LIN {X 0,Y 155.826,Z 845.987,A -85,B 0,C 180,E1 -23873.947,E2 -23873.947} C_VEL
LIN {X 0,Y 159.588,Z 842.317,A -85,B 0,C 180,E1 -23877.541,E2 -23877.541} C_VEL
LIN {X 0,Y 163.776,Z 837.68,A -85,B 0,C 180,E1 -23880.992,E2 -23880.992} C_VEL
LIN {X 0,Y 169.657,Z 830.821,A -85,B 0,C 180,E1 -23884.72,E2 -23884.72} C_VEL
LIN {X 0,Y 175.318,Z 823.487,A -85,B 0,C 180,E1 -23887.684,E2 -23887.684} C_VEL
LIN {X 0,Y 181.515,Z 814.528,A -85,B 0,C 180,E1 -23890.429,E2 -23890.429} C_VEL
LIN {X 0,Y 186.46,Z 805.713,A -85,B 0,C 180,E1 -23892.721,E2 -23892.721} C_VEL
LIN {X 0,Y 191.129,Z 795.722,A -85,B 0,C 180,E1 -23894.904,E2 -23894.904} C_VEL
LIN {X 0,Y 194.213,Z 785.837,A -85,B 0,C 180,E1 -23897.193,E2 -23897.193} C_VEL
LIN {X 0,Y 196.046,Z 776.648,A -85,B 0,C 180,E1 -23899.421,E2 -23899.421} C_VEL
LIN {X 0,Y 196.921,Z 769.856,A -85,B 0,C 180,E1 -23901.188,E2 -23901.188} C_VEL
LIN {X 0,Y 196.991,Z 768.155,A -85,B 0,C 180,E1 -23901.708,E2 -23901.708} C_VEL
LIN {X 0,Y 195.839,Z 762.077,A -85,B 0,C 180,E1 -23904.957,E2 -23904.957} C_VEL
LIN {X 0,Y 195.533,Z 760.977,A -85,B 0,C 180,E1 -23905.757,E2 -23905.757} C_VEL
LIN {X 0,Y 194.784,Z 759.757,A -85,B 0,C 180,E1 -23907.233,E2 -23907.233} C_VEL
LIN {X 0,Y 193.221,Z 757.907,A -85,B 0,C 180,E1 -23911.128,E2 -23911.128} C_VEL
LIN {X 0,Y 192.563,Z 757.534,A -85,B 0,C 180,E1 -23914.025,E2 -23914.025} C_VEL
LIN {X 0,Y 192.277,Z 757.927,A -85,B 0,C 180,E1 -23916.292,E2 -23916.292} C_VEL
LIN {X 0,Y 192.26,Z 758.818,A -85,B 0,C 180,E1 -23918.558,E2 -23918.558} C_VEL
LIN {X 0,Y 192.645,Z 760.564,A -85,B 0,C 180,E1 -23921.531,E2 -23921.531} C_VEL
LIN {X 0,Y 193.16,Z 762.881,A -85,B 0,C 180,E1 -23924.02,E2 -23924.02} C_VEL
LIN {X 0,Y 193.845,Z 765.735,A -85,B 0,C 180,E1 -23926.409,E2 -23926.409} C_VEL
LIN {X 0,Y 194.652,Z 771.052,A -85,B 0,C 180,E1 -23929.599,E2 -23929.599} C_VEL
LIN {X 0,Y 194.221,Z 775.457,A -85,B 0,C 180,E1 -23931.153,E2 -23931.153} C_VEL
LIN {X 0,Y 192.654,Z 785.131,A -85,B 0,C 180,E1 -23934.242,E2 -23934.242} C_VEL
LIN {X 0,Y 190.272,Z 794.462,A -85,B 0,C 180,E1 -23937.142,E2 -23937.142} C_VEL
LIN {X 0,Y 188.258,Z 800.26,A -85,B 0,C 180,E1 -23938.93,E2 -23938.93} C_VEL
LIN {X 0,Y 181.902,Z 810.719,A -85,B 0,C 180,E1 -23941.589,E2 -23941.589} C_VEL
LIN {X 0,Y 175.399,Z 819.674,A -85,B 0,C 180,E1 -23944.596,E2 -23944.596} C_VEL
LIN {X 0,Y 170.121,Z 826.215,A -85,B 0,C 180,E1 -23947.498,E2 -23947.498} C_VEL
LIN {X 0,Y 164.672,Z 832.219,A -85,B 0,C 180,E1 -23951.014,E2 -23951.014} C_VEL
LIN {X 0,Y 159.317,Z 837.423,A -85,B 0,C 180,E1 -23955.348,E2 -23955.348} C_VEL
LIN {X 0,Y 155.916,Z 840.355,A -85,B 0,C 180,E1 -23958.817,E2 -23958.817} C_VEL
LIN {X 0,Y 152.704,Z 842.697,A -85,B 0,C 180,E1 -23963.01,E2 -23963.01} C_VEL
LIN {X 0,Y 149.965,Z 844.066,A -85,B 0,C 180,E1 -23967.946,E2 -23967.946} C_VEL
LIN {X 0,Y 148.566,Z 844.232,A -85,B 0,C 180,E1 -23971.628,E2 -23971.628} C_VEL
LIN {X 0,Y 147.557,Z 843.519,A -85,B 0,C 180,E1 -23975.937,E2 -23975.937} C_VEL
LIN {X 0,Y 147.083,Z 841.894,A -85,B 0,C 180,E1 -23980.139,E2 -23980.139} C_VEL
LIN {X 0,Y 147.203,Z 839.369,A -85,B 0,C 180,E1 -23984.265,E2 -23984.265} C_VEL
LIN {X 0,Y 147.768,Z 835.966,A -85,B 0,C 180,E1 -23988.254,E2 -23988.254} C_VEL
LIN {X 0,Y 148.67,Z 831.692,A -85,B 0,C 180,E1 -23992.083,E2 -23992.083} C_VEL
LIN {X 0,Y 150.258,Z 825.225,A -85,B 0,C 180,E1 -23996.557,E2 -23996.557} C_VEL
LIN {X 0,Y 152.117,Z 818.304,A -85,B 0,C 180,E1 -24000.31,E2 -24000.31} C_VEL
LIN {X 0,Y 154.493,Z 809.866,A -85,B 0,C 180,E1 -24003.95,E2 -24003.95} C_VEL
LIN {X 0,Y 157.066,Z 800.56,A -85,B 0,C 180,E1 -24007.131,E2 -24007.131} C_VEL
LIN {X 0,Y 159.971,Z 789.532,A -85,B 0,C 180,E1 -24010.095,E2 -24010.095} C_VEL
LIN {X 0,Y 162.101,Z 780.609,A -85,B 0,C 180,E1 -24012.008,E2 -24012.008} C_VEL
LIN {X 0,Y 161.942,Z 769.581,A -85,B 0,C 180,E1 -24014.263,E2 -24014.263} C_VEL
LIN {X 0,Y 161.075,Z 757.75,A -85,B 0,C 180,E1 -24016.295,E2 -24016.295} C_VEL
LIN {X 0,Y 159.614,Z 744.505,A -85,B 0,C 180,E1 -24018.114,E2 -24018.114} C_VEL
LIN {X 0,Y 157.757,Z 732.883,A -85,B 0,C 180,E1 -24019.46,E2 -24019.46} C_VEL
LIN {X 0,Y 159.668,Z 724.11,A -85,B 0,C 180,E1 -24024.318,E2 -24024.318} C_VEL
LIN {X 0,Y 159.312,Z 719.069,A -85,B 0,C 180,E1 -24027.473,E2 -24027.473} C_VEL
LIN {X 0,Y 158.489,Z 711.374,A -85,B 0,C 180,E1 -24032.543,E2 -24032.543} C_VEL
LIN {X 0,Y 157.745,Z 708.301,A -85,B 0,C 180,E1 -24034.713,E2 -24034.713} C_VEL
LIN {X 0,Y 161.91,Z 713.53,A -85,B 0,C 180,E1 -24036.857,E2 -24036.857} C_VEL
LIN {X 0,Y 163.628,Z 720.985,A -85,B 0,C 180,E1 -24039.27,E2 -24039.27} C_VEL
LIN {X 0,Y 162.948,Z 724.437,A -85,B 0,C 180,E1 -24040.249,E2 -24040.249} C_VEL
LIN {X 0,Y 160.426,Z 733.712,A -85,B 0,C 180,E1 -24043.16,E2 -24043.16} C_VEL
LIN {X 0,Y 157.619,Z 743.025,A -85,B 0,C 180,E1 -24046.849,E2 -24046.849} C_VEL
LIN {X 0,Y 155.336,Z 750.632,A -85,B 0,C 180,E1 -24050.67,E2 -24050.67} C_VEL
LIN {X 0,Y 153.367,Z 757.474,A -85,B 0,C 180,E1 -24055.081,E2 -24055.081} C_VEL
LIN {X 0,Y 152.207,Z 761.853,A -85,B 0,C 180,E1 -24058.681,E2 -24058.681} C_VEL
LIN {X 0,Y 151.345,Z 766.086,A -85,B 0,C 180,E1 -24063.294,E2 -24063.294} C_VEL
LIN {X 0,Y 151.242,Z 768.983,A -85,B 0,C 180,E1 -24067.818,E2 -24067.818} C_VEL
LIN {X 0,Y 151.842,Z 770.706,A -85,B 0,C 180,E1 -24072.221,E2 -24072.221} C_VEL
LIN {X 0,Y 153.463,Z 771.373,A -85,B 0,C 180,E1 -24077.118,E2 -24077.118} C_VEL
LIN {X 0,Y 155.151,Z 770.994,A -85,B 0,C 180,E1 -24080.642,E2 -24080.642} C_VEL
LIN {X 0,Y 157.614,Z 769.708,A -85,B 0,C 180,E1 -24084.573,E2 -24084.573} C_VEL
LIN {X 0,Y 160.613,Z 767.497,A -85,B 0,C 180,E1 -24088.326,E2 -24088.326} C_VEL
LIN {X 0,Y 164.018,Z 764.381,A -85,B 0,C 180,E1 -24091.879,E2 -24091.879} C_VEL
LIN {X 0,Y 169.07,Z 758.981,A -85,B 0,C 180,E1 -24096.138,E2 -24096.138} C_VEL
LIN {X 0,Y 174.209,Z 752.578,A -85,B 0,C 180,E1 -24099.714,E2 -24099.714} C_VEL
LIN {X 0,Y 179.683,Z 744.584,A -85,B 0,C 180,E1 -24103.073,E2 -24103.073} C_VEL
LIN {X 0,Y 180.22,Z 740.718,A -85,B 0,C 180,E1 -24105.317,E2 -24105.317} C_VEL
LIN {X 0,Y 180.167,Z 735.06,A -85,B 0,C 180,E1 -24108.753,E2 -24108.753} C_VEL
LIN {X 0,Y 179.591,Z 729.771,A -85,B 0,C 180,E1 -24112.128,E2 -24112.128} C_VEL
LIN {X 0,Y 178.743,Z 724.926,A -85,B 0,C 180,E1 -24115.49,E2 -24115.49} C_VEL
LIN {X 0,Y 177.285,Z 719.37,A -85,B 0,C 180,E1 -24120,E2 -24120} C_VEL
LIN {X 0,Y 176.628,Z 716.866,A -85,B 0,C 180,E1 -24122.281,E2 -24122.281} C_VEL
LIN {X 0,Y 175.812,Z 715.036,A -85,B 0,C 180,E1 -24124.586,E2 -24124.586} C_VEL
LIN {X 0,Y 174.96,Z 713.779,A -85,B 0,C 180,E1 -24126.922,E2 -24126.922} C_VEL
LIN {X 0,Y 174.184,Z 713.013,A -85,B 0,C 180,E1 -24129.288,E2 -24129.288} C_VEL
LIN {X 0,Y 172.617,Z 713.732,A -85,B 0,C 180,E1 -24136.559,E2 -24136.559} C_VEL
LIN {X 0,Y 172.623,Z 715.509,A -85,B 0,C 180,E1 -24140.542,E2 -24140.542} C_VEL
LIN {X 0,Y 173.211,Z 719.303,A -85,B 0,C 180,E1 -24145.217,E2 -24145.217} C_VEL
LIN {X 0,Y 174.877,Z 724.229,A -85,B 0,C 180,E1 -24150.072,E2 -24150.072} C_VEL
LIN {X 0,Y 176.562,Z 731.034,A -85,B 0,C 180,E1 -24154.475,E2 -24154.475} C_VEL
LIN {X 0,Y 177.831,Z 737.369,A -85,B 0,C 180,E1 -24157.775,E2 -24157.775} C_VEL
LIN {X 0,Y 178.755,Z 742.992,A -85,B 0,C 180,E1 -24160.37,E2 -24160.37} C_VEL
LIN {X 0,Y 178.012,Z 748.71,A -85,B 0,C 180,E1 -24162.158,E2 -24162.158} C_VEL
LIN {X 0,Y 175.591,Z 759.813,A -85,B 0,C 180,E1 -24165.539,E2 -24165.539} C_VEL
LIN {X 0,Y 172.631,Z 769.223,A -85,B 0,C 180,E1 -24168.586,E2 -24168.586} C_VEL
LIN {X 0,Y 168.859,Z 778.701,A -85,B 0,C 180,E1 -24172.027,E2 -24172.027} C_VEL
LIN {X 0,Y 164.593,Z 786.996,A -85,B 0,C 180,E1 -24175.543,E2 -24175.543} C_VEL
LIN {X 0,Y 160.441,Z 794.744,A -85,B 0,C 180,E1 -24179.75,E2 -24179.75} C_VEL
LIN {X 0,Y 159.775,Z 795.982,A -85,B 0,C 180,E1 -24180.429,E2 -24180.429} C_VEL
LIN {X 0,Y 157.071,Z 806.36,A -85,B 0,C 180,E1 -24183.06,E2 -24183.06} C_VEL
LIN {X 0,Y 154.684,Z 815.135,A -85,B 0,C 180,E1 -24185.862,E2 -24185.862} C_VEL
LIN {X 0,Y 152.114,Z 824.713,A -85,B 0,C 180,E1 -24189.724,E2 -24189.724} C_VEL
LIN {X 0,Y 150.069,Z 832.34,A -85,B 0,C 180,E1 -24193.679,E2 -24193.679} C_VEL
LIN {X 0,Y 148.844,Z 838.458,A -85,B 0,C 180,E1 -24197.731,E2 -24197.731} C_VEL
LIN {X 0,Y 148.118,Z 843.259,A -85,B 0,C 180,E1 -24201.815,E2 -24201.815} C_VEL
LIN {X 0,Y 147.923,Z 845.823,A -85,B 0,C 180,E1 -24204.546,E2 -24204.546} C_VEL
LIN {X 0,Y 147.845,Z 847.879,A -85,B 0,C 180,E1 -24207.274,E2 -24207.274} C_VEL
LIN {X 0,Y 147.968,Z 849.477,A -85,B 0,C 180,E1 -24209.999,E2 -24209.999} C_VEL
LIN {X 0,Y 147.782,Z 851.409,A -85,B 0,C 180,E1 -24215.456,E2 -24215.456} C_VEL
LIN {X 0,Y 148.53,Z 851.738,A -85,B 0,C 180,E1 -24220.909,E2 -24220.909} C_VEL
LIN {X 0,Y 149.722,Z 851.049,A -85,B 0,C 180,E1 -24224.66,E2 -24224.66} C_VEL
LIN {X 0,Y 150.075,Z 850.4,A -85,B 0,C 180,E1 -24226.899,E2 -24226.899} C_VEL
LIN {X 0,Y 149.484,Z 848.906,A -85,B 0,C 180,E1 -24230.641,E2 -24230.641} C_VEL
LIN {X 0,Y 149.352,Z 847.291,A -85,B 0,C 180,E1 -24233.615,E2 -24233.615} C_VEL
LIN {X 0,Y 150.242,Z 845.724,A -85,B 0,C 180,E1 -24235.763,E2 -24235.763} C_VEL
LIN {X 0,Y 150.824,Z 845.125,A -85,B 0,C 180,E1 -24236.44,E2 -24236.44} C_VEL
LIN {X 0,Y 154.632,Z 841.471,A -85,B 0,C 180,E1 -24239.995,E2 -24239.995} C_VEL
LIN {X 0,Y 159.511,Z 836.64,A -85,B 0,C 180,E1 -24243.416,E2 -24243.416} C_VEL
LIN {X 0,Y 165.801,Z 829.618,A -85,B 0,C 180,E1 -24247.157,E2 -24247.157} C_VEL
LIN {X 0,Y 171.98,Z 822.086,A -85,B 0,C 180,E1 -24250.061,E2 -24250.061} C_VEL
LIN {X 0,Y 177.339,Z 814.593,A -85,B 0,C 180,E1 -24252.352,E2 -24252.352} C_VEL
LIN {X 0,Y 183.613,Z 803.967,A -85,B 0,C 180,E1 -24255.079,E2 -24255.079} C_VEL
LIN {X 0,Y 187.168,Z 796.589,A -85,B 0,C 180,E1 -24256.744,E2 -24256.744} C_VEL
LIN {X 0,Y 190.159,Z 788.018,A -85,B 0,C 180,E1 -24258.827,E2 -24258.827} C_VEL
LIN {X 0,Y 192.511,Z 778.595,A -85,B 0,C 180,E1 -24261.25,E2 -24261.25} C_VEL
LIN {X 0,Y 193.42,Z 773.023,A -85,B 0,C 180,E1 -24262.855,E2 -24262.855} C_VEL
LIN {X 0,Y 192.922,Z 768.674,A -85,B 0,C 180,E1 -24265.305,E2 -24265.305} C_VEL
LIN {X 0,Y 192.251,Z 766.491,A -85,B 0,C 180,E1 -24267.222,E2 -24267.222} C_VEL
LIN {X 0,Y 190.756,Z 764.503,A -85,B 0,C 180,E1 -24271.382,E2 -24271.382} C_VEL
LIN {X 0,Y 190.239,Z 764.229,A -85,B 0,C 180,E1 -24273.684,E2 -24273.684} C_VEL
LIN {X 0,Y 189.858,Z 764.532,A -85,B 0,C 180,E1 -24275.971,E2 -24275.971} C_VEL
LIN {X 0,Y 189.762,Z 765.369,A -85,B 0,C 180,E1 -24278.262,E2 -24278.262} C_VEL
LIN {X 0,Y 189.85,Z 766.652,A -85,B 0,C 180,E1 -24280.538,E2 -24280.538} C_VEL
LIN {X 0,Y 190.167,Z 768.348,A -85,B 0,C 180,E1 -24282.803,E2 -24282.803} C_VEL
LIN {X 0,Y 190.47,Z 770.799,A -85,B 0,C 180,E1 -24285.031,E2 -24285.031} C_VEL
LIN {X 0,Y 190.885,Z 775.679,A -85,B 0,C 180,E1 -24288.349,E2 -24288.349} C_VEL
LIN {X 0,Y 190.896,Z 776.713,A -85,B 0,C 180,E1 -24288.871,E2 -24288.871} C_VEL
LIN {X 0,Y 188.97,Z 785.792,A -85,B 0,C 180,E1 -24291.983,E2 -24291.983} C_VEL
LIN {X 0,Y 186.907,Z 793.27,A -85,B 0,C 180,E1 -24294.47,E2 -24294.47} C_VEL
LIN {X 0,Y 183.687,Z 801.818,A -85,B 0,C 180,E1 -24297.265,E2 -24297.265} C_VEL
LIN {X 0,Y 181.19,Z 806.001,A -85,B 0,C 180,E1 -24298.333,E2 -24298.333} C_VEL
LIN {X 0,Y 175.081,Z 814.776,A -85,B 0,C 180,E1 -24300.817,E2 -24300.817} C_VEL
LIN {X 0,Y 169.012,Z 822.359,A -85,B 0,C 180,E1 -24303.661,E2 -24303.661} C_VEL
LIN {X 0,Y 162.863,Z 829.098,A -85,B 0,C 180,E1 -24307.028,E2 -24307.028} C_VEL
LIN {X 0,Y 157.342,Z 834.502,A -85,B 0,C 180,E1 -24310.691,E2 -24310.691} C_VEL
LIN {X 0,Y 152.528,Z 838.658,A -85,B 0,C 180,E1 -24314.629,E2 -24314.629} C_VEL
LIN {X 0,Y 148.022,Z 841.954,A -85,B 0,C 180,E1 -24319.411,E2 -24319.411} C_VEL
LIN {X 0,Y 145.287,Z 843.558,A -85,B 0,C 180,E1 -24323.211,E2 -24323.211} C_VEL
LIN {X 0,Y 142.893,Z 844.432,A -85,B 0,C 180,E1 -24327.715,E2 -24327.715} C_VEL
LIN {X 0,Y 140.976,Z 844.118,A -85,B 0,C 180,E1 -24333.255,E2 -24333.255} C_VEL
LIN {X 0,Y 140.29,Z 843.148,A -85,B 0,C 180,E1 -24336.952,E2 -24336.952} C_VEL
LIN {X 0,Y 140.015,Z 840.25,A -85,B 0,C 180,E1 -24342.759,E2 -24342.759} C_VEL
LIN {X 0,Y 140.432,Z 837.16,A -85,B 0,C 180,E1 -24346.866,E2 -24346.866} C_VEL
LIN {X 0,Y 141.3,Z 832.853,A -85,B 0,C 180,E1 -24351.175,E2 -24351.175} C_VEL
LIN {X 0,Y 142.845,Z 826.534,A -85,B 0,C 180,E1 -24356.003,E2 -24356.003} C_VEL
LIN {X 0,Y 144.732,Z 819.733,A -85,B 0,C 180,E1 -24360.019,E2 -24360.019} C_VEL
LIN {X 0,Y 147.351,Z 810.696,A -85,B 0,C 180,E1 -24364.202,E2 -24364.202} C_VEL
LIN {X 0,Y 150.039,Z 801.278,A -85,B 0,C 180,E1 -24367.632,E2 -24367.632} C_VEL
LIN {X 0,Y 153.26,Z 789.549,A -85,B 0,C 180,E1 -24370.931,E2 -24370.931} C_VEL
LIN {X 0,Y 155.433,Z 780.815,A -85,B 0,C 180,E1 -24372.874,E2 -24372.874} C_VEL
LIN {X 0,Y 155.247,Z 768.754,A -85,B 0,C 180,E1 -24375.426,E2 -24375.426} C_VEL
LIN {X 0,Y 154.241,Z 755.718,A -85,B 0,C 180,E1 -24377.694,E2 -24377.694} C_VEL
LIN {X 0,Y 152.749,Z 742.995,A -85,B 0,C 180,E1 -24379.48,E2 -24379.48} C_VEL
LIN {X 0,Y 151.185,Z 733.073,A -85,B 0,C 180,E1 -24380.638,E2 -24380.638} C_VEL
LIN {X 0,Y 152.87,Z 725.924,A -85,B 0,C 180,E1 -24384.726,E2 -24384.726} C_VEL
LIN {X 0,Y 152.686,Z 721.857,A -85,B 0,C 180,E1 -24387.363,E2 -24387.363} C_VEL
LIN {X 0,Y 151.895,Z 714.015,A -85,B 0,C 180,E1 -24392.653,E2 -24392.653} C_VEL
LIN {X 0,Y 151.429,Z 711.767,A -85,B 0,C 180,E1 -24394.327,E2 -24394.327} C_VEL
LIN {X 0,Y 155.673,Z 717.104,A -85,B 0,C 180,E1 -24396.684,E2 -24396.684} C_VEL
LIN {X 0,Y 156.922,Z 723.03,A -85,B 0,C 180,E1 -24398.745,E2 -24398.745} C_VEL
LIN {X 0,Y 153.85,Z 733.985,A -85,B 0,C 180,E1 -24402.198,E2 -24402.198} C_VEL
LIN {X 0,Y 151.166,Z 742.681,A -85,B 0,C 180,E1 -24405.665,E2 -24405.665} C_VEL
LIN {X 0,Y 148.45,Z 751.289,A -85,B 0,C 180,E1 -24410.075,E2 -24410.075} C_VEL
LIN {X 0,Y 146.535,Z 757.745,A -85,B 0,C 180,E1 -24414.321,E2 -24414.321} C_VEL
LIN {X 0,Y 144.978,Z 763.443,A -85,B 0,C 180,E1 -24419.242,E2 -24419.242} C_VEL
LIN {X 0,Y 144.209,Z 767.53,A -85,B 0,C 180,E1 -24424.056,E2 -24424.056} C_VEL
LIN {X 0,Y 144.315,Z 770.539,A -85,B 0,C 180,E1 -24429.28,E2 -24429.28} C_VEL
LIN {X 0,Y 145.09,Z 771.909,A -85,B 0,C 180,E1 -24433.4,E2 -24433.4} C_VEL
LIN {X 0,Y 146.671,Z 772.451,A -85,B 0,C 180,E1 -24437.869,E2 -24437.869} C_VEL
LIN {X 0,Y 149.437,Z 771.772,A -85,B 0,C 180,E1 -24443.085,E2 -24443.085} C_VEL
LIN {X 0,Y 151.815,Z 770.512,A -85,B 0,C 180,E1 -24446.439,E2 -24446.439} C_VEL
LIN {X 0,Y 156.127,Z 767.287,A -85,B 0,C 180,E1 -24451.391,E2 -24451.391} C_VEL
LIN {X 0,Y 159.839,Z 763.973,A -85,B 0,C 180,E1 -24454.746,E2 -24454.746} C_VEL
LIN {X 0,Y 163.989,Z 759.715,A -85,B 0,C 180,E1 -24457.957,E2 -24457.957} C_VEL
LIN {X 0,Y 168.55,Z 754.391,A -85,B 0,C 180,E1 -24461.013,E2 -24461.013} C_VEL
LIN {X 0,Y 173.841,Z 747.225,A -85,B 0,C 180,E1 -24464.165,E2 -24464.165} C_VEL
LIN {X 0,Y 174.454,Z 744.264,A -85,B 0,C 180,E1 -24466.013,E2 -24466.013} C_VEL
LIN {X 0,Y 174.778,Z 738.941,A -85,B 0,C 180,E1 -24469.575,E2 -24469.575} C_VEL
LIN {X 0,Y 174.538,Z 733.948,A -85,B 0,C 180,E1 -24473.062,E2 -24473.062} C_VEL
LIN {X 0,Y 174.029,Z 729.411,A -85,B 0,C 180,E1 -24476.527,E2 -24476.527} C_VEL
LIN {X 0,Y 173.04,Z 724.266,A -85,B 0,C 180,E1 -24481.164,E2 -24481.164} C_VEL
LIN {X 0,Y 172.836,Z 723.073,A -85,B 0,C 180,E1 -24482.331,E2 -24482.331} C_VEL
LIN {X 0,Y 172.278,Z 721.234,A -85,B 0,C 180,E1 -24484.68,E2 -24484.68} C_VEL
LIN {X 0,Y 171.599,Z 720.018,A -85,B 0,C 180,E1 -24487.058,E2 -24487.058} C_VEL
LIN {X 0,Y 170.921,Z 719.384,A -85,B 0,C 180,E1 -24489.467,E2 -24489.467} C_VEL
LIN {X 0,Y 169.743,Z 719.796,A -85,B 0,C 180,E1 -24494.385,E2 -24494.385} C_VEL
LIN {X 0,Y 169.522,Z 720.566,A -85,B 0,C 180,E1 -24497.533,E2 -24497.533} C_VEL
LIN {X 0,Y 169.548,Z 721.36,A -85,B 0,C 180,E1 -24499.367,E2 -24499.367} C_VEL
LIN {X 0,Y 169.859,Z 725.141,A -85,B 0,C 180,E1 -24504.456,E2 -24504.456} C_VEL
LIN {X 0,Y 170.928,Z 728.993,A -85,B 0,C 180,E1 -24508.569,E2 -24508.569} C_VEL
LIN {X 0,Y 172.085,Z 734.952,A -85,B 0,C 180,E1 -24512.867,E2 -24512.867} C_VEL
LIN {X 0,Y 173.161,Z 741.729,A -85,B 0,C 180,E1 -24516.773,E2 -24516.773} C_VEL
LIN {X 0,Y 173.754,Z 746.744,A -85,B 0,C 180,E1 -24519.257,E2 -24519.257} C_VEL
LIN {X 0,Y 172.743,Z 752.019,A -85,B 0,C 180,E1 -24521.018,E2 -24521.018} C_VEL
LIN {X 0,Y 169.526,Z 763.514,A -85,B 0,C 180,E1 -24524.811,E2 -24524.811} C_VEL
LIN {X 0,Y 165.866,Z 772.924,A -85,B 0,C 180,E1 -24528.136,E2 -24528.136} C_VEL
LIN {X 0,Y 161.709,Z 781.631,A -85,B 0,C 180,E1 -24531.665,E2 -24531.665} C_VEL
LIN {X 0,Y 157.269,Z 789.168,A -85,B 0,C 180,E1 -24535.265,E2 -24535.265} C_VEL
LIN {X 0,Y 152.837,Z 796.671,A -85,B 0,C 180,E1 -24539.804,E2 -24539.804} C_VEL
LIN {X 0,Y 150.017,Z 807.029,A -85,B 0,C 180,E1 -24542.611,E2 -24542.611} C_VEL
LIN {X 0,Y 147.199,Z 816.995,A -85,B 0,C 180,E1 -24546.055,E2 -24546.055} C_VEL
LIN {X 0,Y 145.032,Z 824.748,A -85,B 0,C 180,E1 -24549.43,E2 -24549.43} C_VEL
LIN {X 0,Y 142.953,Z 832.297,A -85,B 0,C 180,E1 -24553.578,E2 -24553.578} C_VEL
LIN {X 0,Y 141.558,Z 839.261,A -85,B 0,C 180,E1 -24558.544,E2 -24558.544} C_VEL
LIN {X 0,Y 140.926,Z 843.832,A -85,B 0,C 180,E1 -24562.837,E2 -24562.837} C_VEL
LIN {X 0,Y 140.777,Z 847.259,A -85,B 0,C 180,E1 -24567.137,E2 -24567.137} C_VEL
LIN {X 0,Y 140.891,Z 848.958,A -85,B 0,C 180,E1 -24569.998,E2 -24569.998} C_VEL
LIN {X 0,Y 140.709,Z 851.029,A -85,B 0,C 180,E1 -24575.732,E2 -24575.732} C_VEL
LIN {X 0,Y 141.532,Z 851.57,A -85,B 0,C 180,E1 -24581.455,E2 -24581.455} C_VEL
LIN {X 0,Y 143.572,Z 850.578,A -85,B 0,C 180,E1 -24587.078,E2 -24587.078} C_VEL
LIN {X 0,Y 147.048,Z 848.132,A -85,B 0,C 180,E1 -24592.478,E2 -24592.478} C_VEL
LIN {X 0,Y 150.824,Z 845.125,A -85,B 0,C 180,E1 -24596.44,E2 -24596.44} C_VEL
LIN {X 0,Y 151.56,Z 843.941,A -85,B 0,C 180,E1 -24597.861,E2 -24597.861} C_VEL
LIN {X 0,Y 151.222,Z 840.124,A -85,B 0,C 180,E1 -24602.774,E2 -24602.774} C_VEL
LIN {X 0,Y 152.404,Z 838.576,A -85,B 0,C 180,E1 -24604.078,E2 -24604.078} C_VEL
LIN {X 0,Y 158.309,Z 832.799,A -85,B 0,C 180,E1 -24607.618,E2 -24607.618} C_VEL
LIN {X 0,Y 164.454,Z 826.042,A -85,B 0,C 180,E1 -24610.669,E2 -24610.669} C_VEL
LIN {X 0,Y 171.225,Z 817.803,A -85,B 0,C 180,E1 -24613.431,E2 -24613.431} C_VEL
LIN {X 0,Y 177.764,Z 808.035,A -85,B 0,C 180,E1 -24616.178,E2 -24616.178} C_VEL
LIN {X 0,Y 182.644,Z 799.271,A -85,B 0,C 180,E1 -24618.227,E2 -24618.227} C_VEL
LIN {X 0,Y 186.284,Z 790.329,A -85,B 0,C 180,E1 -24620.502,E2 -24620.502} C_VEL
LIN {X 0,Y 188.724,Z 782.307,A -85,B 0,C 180,E1 -24622.671,E2 -24622.671} C_VEL
LIN {X 0,Y 189.549,Z 779.002,A -85,B 0,C 180,E1 -24623.612,E2 -24623.612} C_VEL
LIN {X 0,Y 189.755,Z 777.557,A -85,B 0,C 180,E1 -24624.151,E2 -24624.151} C_VEL
LIN {X 0,Y 189.6,Z 774.282,A -85,B 0,C 180,E1 -24626.219,E2 -24626.219} C_VEL
LIN {X 0,Y 189.278,Z 772.88,A -85,B 0,C 180,E1 -24627.467,E2 -24627.467} C_VEL
LIN {X 0,Y 188.109,Z 771.241,A -85,B 0,C 180,E1 -24630.941,E2 -24630.941} C_VEL
LIN {X 0,Y 187.39,Z 770.843,A -85,B 0,C 180,E1 -24634.169,E2 -24634.169} C_VEL
LIN {X 0,Y 186.953,Z 771.779,A -85,B 0,C 180,E1 -24637.918,E2 -24637.918} C_VEL
LIN {X 0,Y 186.898,Z 773.008,A -85,B 0,C 180,E1 -24640.218,E2 -24640.218} C_VEL
LIN {X 0,Y 187.025,Z 774.687,A -85,B 0,C 180,E1 -24642.505,E2 -24642.505} C_VEL
LIN {X 0,Y 187.106,Z 777.126,A -85,B 0,C 180,E1 -24644.756,E2 -24644.756} C_VEL
LIN {X 0,Y 187.068,Z 781.229,A -85,B 0,C 180,E1 -24647.627,E2 -24647.627} C_VEL
LIN {X 0,Y 185.194,Z 788.135,A -85,B 0,C 180,E1 -24650.167,E2 -24650.167} C_VEL
LIN {X 0,Y 182.669,Z 795.636,A -85,B 0,C 180,E1 -24652.817,E2 -24652.817} C_VEL
LIN {X 0,Y 179.344,Z 803.462,A -85,B 0,C 180,E1 -24655.505,E2 -24655.505} C_VEL
LIN {X 0,Y 177.894,Z 805.885,A -85,B 0,C 180,E1 -24656.211,E2 -24656.211} C_VEL
LIN {X 0,Y 171.284,Z 814.896,A -85,B 0,C 180,E1 -24658.74,E2 -24658.74} C_VEL
LIN {X 0,Y 164.245,Z 823.121,A -85,B 0,C 180,E1 -24661.839,E2 -24661.839} C_VEL
LIN {X 0,Y 157.99,Z 829.554,A -85,B 0,C 180,E1 -24665.104,E2 -24665.104} C_VEL
LIN {X 0,Y 151.688,Z 835.248,A -85,B 0,C 180,E1 -24669.102,E2 -24669.102} C_VEL
LIN {X 0,Y 145.644,Z 839.863,A -85,B 0,C 180,E1 -24673.961,E2 -24673.961} C_VEL
LIN {X 0,Y 141.084,Z 842.765,A -85,B 0,C 180,E1 -24678.837,E2 -24678.837} C_VEL
LIN {X 0,Y 137.444,Z 844.386,A -85,B 0,C 180,E1 -24684.146,E2 -24684.146} C_VEL
LIN {X 0,Y 135.496,Z 844.71,A -85,B 0,C 180,E1 -24688.148,E2 -24688.148} C_VEL
LIN {X 0,Y 133.947,Z 844.193,A -85,B 0,C 180,E1 -24692.917,E2 -24692.917} C_VEL
LIN {X 0,Y 133.109,Z 842.739,A -85,B 0,C 180,E1 -24697.632,E2 -24697.632} C_VEL
LIN {X 0,Y 132.971,Z 839.668,A -85,B 0,C 180,E1 -24703.4,E2 -24703.4} C_VEL
LIN {X 0,Y 133.432,Z 836.52,A -85,B 0,C 180,E1 -24707.51,E2 -24707.51} C_VEL
LIN {X 0,Y 134.524,Z 831.349,A -85,B 0,C 180,E1 -24712.574,E2 -24712.574} C_VEL
LIN {X 0,Y 136.343,Z 824.55,A -85,B 0,C 180,E1 -24717.587,E2 -24717.587} C_VEL
LIN {X 0,Y 138.549,Z 816.793,A -85,B 0,C 180,E1 -24722.019,E2 -24722.019} C_VEL
LIN {X 0,Y 141.344,Z 807.558,A -85,B 0,C 180,E1 -24726.103,E2 -24726.103} C_VEL
LIN {X 0,Y 144.146,Z 798.158,A -85,B 0,C 180,E1 -24729.39,E2 -24729.39} C_VEL
LIN {X 0,Y 146.843,Z 788.49,A -85,B 0,C 180,E1 -24732.082,E2 -24732.082} C_VEL
LIN {X 0,Y 148.74,Z 780.586,A -85,B 0,C 180,E1 -24733.885,E2 -24733.885} C_VEL
LIN {X 0,Y 148.599,Z 769.646,A -85,B 0,C 180,E1 -24736.323,E2 -24736.323} C_VEL
LIN {X 0,Y 147.736,Z 756.887,A -85,B 0,C 180,E1 -24738.685,E2 -24738.685} C_VEL
LIN {X 0,Y 146.354,Z 744.277,A -85,B 0,C 180,E1 -24740.587,E2 -24740.587} C_VEL
LIN {X 0,Y 144.682,Z 733.207,A -85,B 0,C 180,E1 -24741.974,E2 -24741.974} C_VEL
LIN {X 0,Y 146.197,Z 726.664,A -85,B 0,C 180,E1 -24745.866,E2 -24745.866} C_VEL
LIN {X 0,Y 145.447,Z 718.668,A -85,B 0,C 180,E1 -24751.386,E2 -24751.386} C_VEL
LIN {X 0,Y 145.059,Z 715.17,A -85,B 0,C 180,E1 -24753.908,E2 -24753.908} C_VEL
LIN {X 0,Y 149.241,Z 720.362,A -85,B 0,C 180,E1 -24756.402,E2 -24756.402} C_VEL
LIN {X 0,Y 149.982,Z 723.305,A -85,B 0,C 180,E1 -24757.511,E2 -24757.511} C_VEL
LIN {X 0,Y 150.082,Z 724.864,A -85,B 0,C 180,E1 -24758.077,E2 -24758.077} C_VEL
LIN {X 0,Y 147.134,Z 734.848,A -85,B 0,C 180,E1 -24761.365,E2 -24761.365} C_VEL
LIN {X 0,Y 144.448,Z 743.194,A -85,B 0,C 180,E1 -24764.799,E2 -24764.799} C_VEL
LIN {X 0,Y 142.229,Z 750.018,A -85,B 0,C 180,E1 -24768.285,E2 -24768.285} C_VEL
LIN {X 0,Y 139.941,Z 757.179,A -85,B 0,C 180,E1 -24772.907,E2 -24772.907} C_VEL
LIN {X 0,Y 138.43,Z 762.365,A -85,B 0,C 180,E1 -24777.19,E2 -24777.19} C_VEL
LIN {X 0,Y 137.307,Z 767.245,A -85,B 0,C 180,E1 -24782.511,E2 -24782.511} C_VEL
LIN {X 0,Y 137.171,Z 770.707,A -85,B 0,C 180,E1 -24787.941,E2 -24787.941} C_VEL
LIN {X 0,Y 137.622,Z 772.243,A -85,B 0,C 180,E1 -24791.598,E2 -24791.598} C_VEL
LIN {X 0,Y 138.578,Z 773.192,A -85,B 0,C 180,E1 -24795.238,E2 -24795.238} C_VEL
LIN {X 0,Y 140.23,Z 773.548,A -85,B 0,C 180,E1 -24799.344,E2 -24799.344} C_VEL
LIN {X 0,Y 142.672,Z 773.015,A -85,B 0,C 180,E1 -24803.764,E2 -24803.764} C_VEL
LIN {X 0,Y 145.736,Z 771.551,A -85,B 0,C 180,E1 -24807.963,E2 -24807.963} C_VEL
LIN {X 0,Y 150.15,Z 768.519,A -85,B 0,C 180,E1 -24812.79,E2 -24812.79} C_VEL
LIN {X 0,Y 153.844,Z 765.492,A -85,B 0,C 180,E1 -24816.017,E2 -24816.017} C_VEL
LIN {X 0,Y 159.046,Z 760.459,A -85,B 0,C 180,E1 -24819.884,E2 -24819.884} C_VEL
LIN {X 0,Y 164.905,Z 753.86,A -85,B 0,C 180,E1 -24823.563,E2 -24823.563} C_VEL
LIN {X 0,Y 168.285,Z 749.563,A -85,B 0,C 180,E1 -24825.489,E2 -24825.489} C_VEL
LIN {X 0,Y 168.953,Z 746.067,A -85,B 0,C 180,E1 -24827.996,E2 -24827.996} C_VEL
LIN {X 0,Y 169.397,Z 741.125,A -85,B 0,C 180,E1 -24831.651,E2 -24831.651} C_VEL
LIN {X 0,Y 169.394,Z 736.593,A -85,B 0,C 180,E1 -24835.241,E2 -24835.241} C_VEL
LIN {X 0,Y 169.105,Z 732.593,A -85,B 0,C 180,E1 -24838.81,E2 -24838.81} C_VEL
LIN {X 0,Y 168.755,Z 729.069,A -85,B 0,C 180,E1 -24842.387,E2 -24842.387} C_VEL
LIN {X 0,Y 168.437,Z 727.254,A -85,B 0,C 180,E1 -24844.787,E2 -24844.787} C_VEL
LIN {X 0,Y 167.916,Z 726.073,A -85,B 0,C 180,E1 -24847.214,E2 -24847.214} C_VEL
LIN {X 0,Y 167.347,Z 725.581,A -85,B 0,C 180,E1 -24849.671,E2 -24849.671} C_VEL
LIN {X 0,Y 166.304,Z 726.111,A -85,B 0,C 180,E1 -24854.689,E2 -24854.689} C_VEL
LIN {X 0,Y 166.139,Z 726.742,A -85,B 0,C 180,E1 -24857.225,E2 -24857.225} C_VEL
LIN {X 0,Y 166.072,Z 729.064,A -85,B 0,C 180,E1 -24861.404,E2 -24861.404} C_VEL
LIN {X 0,Y 167.022,Z 734.621,A -85,B 0,C 180,E1 -24867.913,E2 -24867.913} C_VEL
LIN {X 0,Y 167.744,Z 740.139,A -85,B 0,C 180,E1 -24872.129,E2 -24872.129} C_VEL
LIN {X 0,Y 168.367,Z 746.054,A -85,B 0,C 180,E1 -24875.76,E2 -24875.76} C_VEL
LIN {X 0,Y 168.608,Z 750.801,A -85,B 0,C 180,E1 -24878.295,E2 -24878.295} C_VEL
LIN {X 0,Y 166.057,Z 759.504,A -85,B 0,C 180,E1 -24881.303,E2 -24881.303} C_VEL
LIN {X 0,Y 162.974,Z 767.713,A -85,B 0,C 180,E1 -24884.286,E2 -24884.286} C_VEL
LIN {X 0,Y 159.053,Z 776.24,A -85,B 0,C 180,E1 -24887.634,E2 -24887.634} C_VEL
LIN {X 0,Y 154.502,Z 784.303,A -85,B 0,C 180,E1 -24891.283,E2 -24891.283} C_VEL
LIN {X 0,Y 149.322,Z 792.061,A -85,B 0,C 180,E1 -24895.611,E2 -24895.611} C_VEL
LIN {X 0,Y 145.919,Z 797.096,A -85,B 0,C 180,E1 -24899.118,E2 -24899.118} C_VEL
LIN {X 0,Y 142.763,Z 808.371,A -85,B 0,C 180,E1 -24902.39,E2 -24902.39} C_VEL
LIN {X 0,Y 140.193,Z 817.001,A -85,B 0,C 180,E1 -24905.569,E2 -24905.569} C_VEL
LIN {X 0,Y 137.963,Z 824.717,A -85,B 0,C 180,E1 -24909.108,E2 -24909.108} C_VEL
LIN {X 0,Y 135.835,Z 832.225,A -85,B 0,C 180,E1 -24913.466,E2 -24913.466} C_VEL
LIN {X 0,Y 134.595,Z 838.269,A -85,B 0,C 180,E1 -24917.943,E2 -24917.943} C_VEL
LIN {X 0,Y 133.892,Z 843.009,A -85,B 0,C 180,E1 -24922.458,E2 -24922.458} C_VEL
LIN {X 0,Y 133.718,Z 846.589,A -85,B 0,C 180,E1 -24926.986,E2 -24926.986} C_VEL
LIN {X 0,Y 133.816,Z 848.399,A -85,B 0,C 180,E1 -24929.998,E2 -24929.998} C_VEL
LIN {X 0,Y 133.598,Z 849.72,A -85,B 0,C 180,E1 -24933.014,E2 -24933.014} C_VEL
LIN {X 0,Y 133.956,Z 851.173,A -85,B 0,C 180,E1 -24939.054,E2 -24939.054} C_VEL
LIN {X 0,Y 135.508,Z 851.157,A -85,B 0,C 180,E1 -24945.028,E2 -24945.028} C_VEL
LIN {X 0,Y 138.42,Z 849.621,A -85,B 0,C 180,E1 -24950.817,E2 -24950.817} C_VEL
LIN {X 0,Y 142.973,Z 846.62,A -85,B 0,C 180,E1 -24956.256,E2 -24956.256} C_VEL
LIN {X 0,Y 147.122,Z 843.308,A -85,B 0,C 180,E1 -24960.103,E2 -24960.103} C_VEL
LIN {X 0,Y 152.404,Z 838.576,A -85,B 0,C 180,E1 -24964.078,E2 -24964.078} C_VEL
LIN {X 0,Y 154.62,Z 836.104,A -85,B 0,C 180,E1 -24965.901,E2 -24965.901} C_VEL
LIN {X 0,Y 156.946,Z 831.937,A -85,B 0,C 180,E1 -24969.109,E2 -24969.109} C_VEL
LIN {X 0,Y 159.645,Z 827.299,A -85,B 0,C 180,E1 -24972.108,E2 -24972.108} C_VEL
LIN {X 0,Y 162.322,Z 824.013,A -85,B 0,C 180,E1 -24973.558,E2 -24973.558} C_VEL
LIN {X 0,Y 168.521,Z 816.525,A -85,B 0,C 180,E1 -24976.002,E2 -24976.002} C_VEL
LIN {X 0,Y 175.409,Z 806.543,A -85,B 0,C 180,E1 -24978.696,E2 -24978.696} C_VEL
LIN {X 0,Y 178.772,Z 800.823,A -85,B 0,C 180,E1 -24980.07,E2 -24980.07} C_VEL
LIN {X 0,Y 182.828,Z 791.896,A -85,B 0,C 180,E1 -24982.447,E2 -24982.447} C_VEL
LIN {X 0,Y 185.762,Z 783.628,A -85,B 0,C 180,E1 -24984.844,E2 -24984.844} C_VEL
LIN {X 0,Y 186.053,Z 782.133,A -85,B 0,C 180,E1 -24985.485,E2 -24985.485} C_VEL
LIN {X 0,Y 186.088,Z 780.128,A -85,B 0,C 180,E1 -24986.838,E2 -24986.838} C_VEL
LIN {X 0,Y 185.879,Z 778.937,A -85,B 0,C 180,E1 -24988.039,E2 -24988.039} C_VEL
LIN {X 0,Y 185.033,Z 777.683,A -85,B 0,C 180,E1 -24990.876,E2 -24990.876} C_VEL
LIN {X 0,Y 184.585,Z 777.273,A -85,B 0,C 180,E1 -24992.813,E2 -24992.813} C_VEL
LIN {X 0,Y 184.137,Z 777.355,A -85,B 0,C 180,E1 -24995.175,E2 -24995.175} C_VEL
LIN {X 0,Y 183.835,Z 778.048,A -85,B 0,C 180,E1 -24997.523,E2 -24997.523} C_VEL
LIN {X 0,Y 183.614,Z 779.192,A -85,B 0,C 180,E1 -24999.849,E2 -24999.849} C_VEL
LIN {X 0,Y 183.584,Z 780.84,A -85,B 0,C 180,E1 -25002.166,E2 -25002.166} C_VEL
LIN {X 0,Y 183.283,Z 784.687,A -85,B 0,C 180,E1 -25005.567,E2 -25005.567} C_VEL
LIN {X 0,Y 183.067,Z 786.398,A -85,B 0,C 180,E1 -25006.682,E2 -25006.682} C_VEL
LIN {X 0,Y 179.986,Z 794.752,A -85,B 0,C 180,E1 -25009.879,E2 -25009.879} C_VEL
LIN {X 0,Y 176.69,Z 802.087,A -85,B 0,C 180,E1 -25012.563,E2 -25012.563} C_VEL
LIN {X 0,Y 174.262,Z 806.628,A -85,B 0,C 180,E1 -25014.213,E2 -25014.213} C_VEL
LIN {X 0,Y 167.456,Z 815.45,A -85,B 0,C 180,E1 -25016.68,E2 -25016.68} C_VEL
LIN {X 0,Y 160.847,Z 822.781,A -85,B 0,C 180,E1 -25019.389,E2 -25019.389} C_VEL
LIN {X 0,Y 154.18,Z 829.254,A -85,B 0,C 180,E1 -25022.612,E2 -25022.612} C_VEL
LIN {X 0,Y 146.692,Z 835.581,A -85,B 0,C 180,E1 -25027.029,E2 -25027.029} C_VEL
LIN {X 0,Y 140.684,Z 839.833,A -85,B 0,C 180,E1 -25031.526,E2 -25031.526} C_VEL
LIN {X 0,Y 137.136,Z 841.996,A -85,B 0,C 180,E1 -25034.847,E2 -25034.847} C_VEL
LIN {X 0,Y 133.647,Z 843.705,A -85,B 0,C 180,E1 -25038.824,E2 -25038.824} C_VEL
LIN {X 0,Y 130.444,Z 844.77,A -85,B 0,C 180,E1 -25043.669,E2 -25043.669} C_VEL
LIN {X 0,Y 127.712,Z 844.747,A -85,B 0,C 180,E1 -25049.687,E2 -25049.687} C_VEL
LIN {X 0,Y 126.633,Z 843.921,A -85,B 0,C 180,E1 -25053.71,E2 -25053.71} C_VEL
LIN {X 0,Y 125.901,Z 842.125,A -85,B 0,C 180,E1 -25058.605,E2 -25058.605} C_VEL
LIN {X 0,Y 125.878,Z 839.405,A -85,B 0,C 180,E1 -25063.466,E2 -25063.466} C_VEL
LIN {X 0,Y 126.647,Z 834.72,A -85,B 0,C 180,E1 -25069.37,E2 -25069.37} C_VEL
LIN {X 0,Y 127.841,Z 829.67,A -85,B 0,C 180,E1 -25074.092,E2 -25074.092} C_VEL
LIN {X 0,Y 129.869,Z 822.521,A -85,B 0,C 180,E1 -25079.229,E2 -25079.229} C_VEL
LIN {X 0,Y 132.212,Z 814.693,A -85,B 0,C 180,E1 -25083.62,E2 -25083.62} C_VEL
LIN {X 0,Y 134.888,Z 806.191,A -85,B 0,C 180,E1 -25087.397,E2 -25087.397} C_VEL
LIN {X 0,Y 138.132,Z 795.543,A -85,B 0,C 180,E1 -25091.075,E2 -25091.075} C_VEL
LIN {X 0,Y 141.374,Z 784.07,A -85,B 0,C 180,E1 -25094.134,E2 -25094.134} C_VEL
LIN {X 0,Y 142.026,Z 780.58,A -85,B 0,C 180,E1 -25094.944,E2 -25094.944} C_VEL
LIN {X 0,Y 141.945,Z 769.673,A -85,B 0,C 180,E1 -25097.491,E2 -25097.491} C_VEL
LIN {X 0,Y 141.153,Z 756.812,A -85,B 0,C 180,E1 -25099.966,E2 -25099.966} C_VEL
LIN {X 0,Y 139.883,Z 744.634,A -85,B 0,C 180,E1 -25101.878,E2 -25101.878} C_VEL
LIN {X 0,Y 138.248,Z 733.231,A -85,B 0,C 180,E1 -25103.434,E2 -25103.434} C_VEL
LIN {X 0,Y 139.441,Z 728.454,A -85,B 0,C 180,E1 -25106.389,E2 -25106.389} C_VEL
LIN {X 0,Y 138.692,Z 719.401,A -85,B 0,C 180,E1 -25112.906,E2 -25112.906} C_VEL
LIN {X 0,Y 138.641,Z 718.644,A -85,B 0,C 180,E1 -25113.544,E2 -25113.544} C_VEL
LIN {X 0,Y 142.705,Z 723.508,A -85,B 0,C 180,E1 -25116.099,E2 -25116.099} C_VEL
LIN {X 0,Y 143.392,Z 725.708,A -85,B 0,C 180,E1 -25117.033,E2 -25117.033} C_VEL
LIN {X 0,Y 140.455,Z 735.631,A -85,B 0,C 180,E1 -25120.452,E2 -25120.452} C_VEL
LIN {X 0,Y 137.634,Z 743.984,A -85,B 0,C 180,E1 -25124.024,E2 -25124.024} C_VEL
LIN {X 0,Y 135.018,Z 751.72,A -85,B 0,C 180,E1 -25128.2,E2 -25128.2} C_VEL
LIN {X 0,Y 132.606,Z 759.143,A -85,B 0,C 180,E1 -25133.386,E2 -25133.386} C_VEL
LIN {X 0,Y 130.885,Z 765.116,A -85,B 0,C 180,E1 -25138.901,E2 -25138.901} C_VEL
LIN {X 0,Y 130.086,Z 769.334,A -85,B 0,C 180,E1 -25144.259,E2 -25144.259} C_VEL
LIN {X 0,Y 130.341,Z 772.587,A -85,B 0,C 180,E1 -25150.321,E2 -25150.321} C_VEL
LIN {X 0,Y 131.765,Z 774.262,A -85,B 0,C 180,E1 -25156.102,E2 -25156.102} C_VEL
LIN {X 0,Y 134.282,Z 774.565,A -85,B 0,C 180,E1 -25161.728,E2 -25161.728} C_VEL
LIN {X 0,Y 136.607,Z 774.012,A -85,B 0,C 180,E1 -25165.535,E2 -25165.535} C_VEL
LIN {X 0,Y 139.988,Z 772.483,A -85,B 0,C 180,E1 -25169.865,E2 -25169.865} C_VEL
LIN {X 0,Y 143.856,Z 770.058,A -85,B 0,C 180,E1 -25173.916,E2 -25173.916} C_VEL
LIN {X 0,Y 148.369,Z 766.64,A -85,B 0,C 180,E1 -25177.732,E2 -25177.732} C_VEL
LIN {X 0,Y 153.367,Z 762.213,A -85,B 0,C 180,E1 -25181.291,E2 -25181.291} C_VEL
LIN {X 0,Y 158.725,Z 756.702,A -85,B 0,C 180,E1 -25184.594,E2 -25184.594} C_VEL
LIN {X 0,Y 162.133,Z 752.745,A -85,B 0,C 180,E1 -25186.475,E2 -25186.475} C_VEL
LIN {X 0,Y 162.897,Z 751.159,A -85,B 0,C 180,E1 -25187.543,E2 -25187.543} C_VEL
LIN {X 0,Y 163.843,Z 746.418,A -85,B 0,C 180,E1 -25191.365,E2 -25191.365} C_VEL
LIN {X 0,Y 164.298,Z 742.067,A -85,B 0,C 180,E1 -25195.093,E2 -25195.093} C_VEL
LIN {X 0,Y 164.409,Z 738.205,A -85,B 0,C 180,E1 -25198.776,E2 -25198.776} C_VEL
LIN {X 0,Y 164.393,Z 734.846,A -85,B 0,C 180,E1 -25202.451,E2 -25202.451} C_VEL
LIN {X 0,Y 164.305,Z 733.081,A -85,B 0,C 180,E1 -25204.908,E2 -25204.908} C_VEL
LIN {X 0,Y 163.943,Z 731.955,A -85,B 0,C 180,E1 -25207.389,E2 -25207.389} C_VEL
LIN {X 0,Y 163.457,Z 731.583,A -85,B 0,C 180,E1 -25209.904,E2 -25209.904} C_VEL
LIN {X 0,Y 162.542,Z 732.279,A -85,B 0,C 180,E1 -25215.037,E2 -25215.037} C_VEL
LIN {X 0,Y 162.365,Z 733.156,A -85,B 0,C 180,E1 -25217.77,E2 -25217.77} C_VEL
LIN {X 0,Y 162.286,Z 734.499,A -85,B 0,C 180,E1 -25220.271,E2 -25220.271} C_VEL
LIN {X 0,Y 162.54,Z 738.65,A -85,B 0,C 180,E1 -25225.62,E2 -25225.62} C_VEL
LIN {X 0,Y 162.947,Z 741.23,A -85,B 0,C 180,E1 -25228.323,E2 -25228.323} C_VEL
LIN {X 0,Y 163.307,Z 746.198,A -85,B 0,C 180,E1 -25232.136,E2 -25232.136} C_VEL
LIN {X 0,Y 163.476,Z 754.074,A -85,B 0,C 180,E1 -25237.005,E2 -25237.005} C_VEL
LIN {X 0,Y 160.579,Z 762.128,A -85,B 0,C 180,E1 -25240.01,E2 -25240.01} C_VEL
LIN {X 0,Y 157.283,Z 769.611,A -85,B 0,C 180,E1 -25242.927,E2 -25242.927} C_VEL
LIN {X 0,Y 152.933,Z 777.804,A -85,B 0,C 180,E1 -25246.422,E2 -25246.422} C_VEL
LIN {X 0,Y 148.108,Z 785.405,A -85,B 0,C 180,E1 -25250.162,E2 -25250.162} C_VEL
LIN {X 0,Y 143.374,Z 791.75,A -85,B 0,C 180,E1 -25253.967,E2 -25253.967} C_VEL
LIN {X 0,Y 139.021,Z 797.5,A -85,B 0,C 180,E1 -25258.364,E2 -25258.364} C_VEL
LIN {X 0,Y 135.784,Z 808.616,A -85,B 0,C 180,E1 -25261.766,E2 -25261.766} C_VEL
LIN {X 0,Y 133.191,Z 817.005,A -85,B 0,C 180,E1 -25265.029,E2 -25265.029} C_VEL
LIN {X 0,Y 130.511,Z 826.018,A -85,B 0,C 180,E1 -25269.51,E2 -25269.51} C_VEL
LIN {X 0,Y 128.469,Z 833.227,A -85,B 0,C 180,E1 -25274.124,E2 -25274.124} C_VEL
LIN {X 0,Y 127.316,Z 839.018,A -85,B 0,C 180,E1 -25278.859,E2 -25278.859} C_VEL
LIN {X 0,Y 126.725,Z 843.525,A -85,B 0,C 180,E1 -25283.63,E2 -25283.63} C_VEL
LIN {X 0,Y 126.659,Z 846.109,A -85,B 0,C 180,E1 -25287.176,E2 -25287.176} C_VEL
LIN {X 0,Y 126.742,Z 847.769,A -85,B 0,C 180,E1 -25289.998,E2 -25289.998} C_VEL
LIN {X 0,Y 126.537,Z 849.202,A -85,B 0,C 180,E1 -25293.182,E2 -25293.182} C_VEL
LIN {X 0,Y 126.568,Z 850.233,A -85,B 0,C 180,E1 -25296.374,E2 -25296.374} C_VEL
LIN {X 0,Y 127.609,Z 851.103,A -85,B 0,C 180,E1 -25302.725,E2 -25302.725} C_VEL
LIN {X 0,Y 129.995,Z 850.538,A -85,B 0,C 180,E1 -25308.926,E2 -25308.926} C_VEL
LIN {X 0,Y 131.806,Z 849.708,A -85,B 0,C 180,E1 -25311.914,E2 -25311.914} C_VEL
LIN {X 0,Y 136.638,Z 846.892,A -85,B 0,C 180,E1 -25317.574,E2 -25317.574} C_VEL
LIN {X 0,Y 142.565,Z 842.594,A -85,B 0,C 180,E1 -25322.836,E2 -25322.836} C_VEL
LIN {X 0,Y 147.967,Z 838.206,A -85,B 0,C 180,E1 -25326.419,E2 -25326.419} C_VEL
LIN {X 0,Y 154.848,Z 831.748,A -85,B 0,C 180,E1 -25330.295,E2 -25330.295} C_VEL
LIN {X 0,Y 161.529,Z 824.864,A -85,B 0,C 180,E1 -25333.255,E2 -25333.255} C_VEL
LIN {X 0,Y 162.322,Z 824.013,A -85,B 0,C 180,E1 -25333.558,E2 -25333.558} C_VEL
LIN {X 0,Y 165.061,Z 820.595,A -85,B 0,C 180,E1 -25334.94,E2 -25334.94} C_VEL
LIN {X 0,Y 168.169,Z 815.069,A -85,B 0,C 180,E1 -25337.558,E2 -25337.558} C_VEL
LIN {X 0,Y 171.103,Z 809.151,A -85,B 0,C 180,E1 -25340.084,E2 -25340.084} C_VEL
LIN {X 0,Y 173.481,Z 805.107,A -85,B 0,C 180,E1 -25341.298,E2 -25341.298} C_VEL
LIN {X 0,Y 177.609,Z 797.731,A -85,B 0,C 180,E1 -25343.278,E2 -25343.278} C_VEL
LIN {X 0,Y 180.313,Z 791.979,A -85,B 0,C 180,E1 -25344.933,E2 -25344.933} C_VEL
LIN {X 0,Y 181.983,Z 787.91,A -85,B 0,C 180,E1 -25346.187,E2 -25346.187} C_VEL
LIN {X 0,Y 182.219,Z 786.97,A -85,B 0,C 180,E1 -25346.632,E2 -25346.632} C_VEL
LIN {X 0,Y 182.28,Z 785.289,A -85,B 0,C 180,E1 -25348.017,E2 -25348.017} C_VEL
LIN {X 0,Y 181.857,Z 784.335,A -85,B 0,C 180,E1 -25349.841,E2 -25349.841} C_VEL
LIN {X 0,Y 181.117,Z 783.511,A -85,B 0,C 180,E1 -25353.184,E2 -25353.184} C_VEL
LIN {X 0,Y 180.398,Z 784.107,A -85,B 0,C 180,E1 -25357.071,E2 -25357.071} C_VEL
LIN {X 0,Y 180.065,Z 785.219,A -85,B 0,C 180,E1 -25359.505,E2 -25359.505} C_VEL
LIN {X 0,Y 179.853,Z 786.8,A -85,B 0,C 180,E1 -25361.783,E2 -25361.783} C_VEL
LIN {X 0,Y 179.409,Z 789.139,A -85,B 0,C 180,E1 -25364.085,E2 -25364.085} C_VEL
LIN {X 0,Y 179.116,Z 790.622,A -85,B 0,C 180,E1 -25365.224,E2 -25365.224} C_VEL
LIN {X 0,Y 178.25,Z 792.914,A -85,B 0,C 180,E1 -25366.316,E2 -25366.316} C_VEL
LIN {X 0,Y 173.968,Z 801.794,A -85,B 0,C 180,E1 -25369.82,E2 -25369.82} C_VEL
LIN {X 0,Y 170.19,Z 808.418,A -85,B 0,C 180,E1 -25372.33,E2 -25372.33} C_VEL
LIN {X 0,Y 162.223,Z 817.844,A -85,B 0,C 180,E1 -25375.137,E2 -25375.137} C_VEL
LIN {X 0,Y 154.691,Z 825.445,A -85,B 0,C 180,E1 -25378.155,E2 -25378.155} C_VEL
LIN {X 0,Y 147.636,Z 831.589,A -85,B 0,C 180,E1 -25381.537,E2 -25381.537} C_VEL
LIN {X 0,Y 140.452,Z 836.939,A -85,B 0,C 180,E1 -25385.743,E2 -25385.743} C_VEL
LIN {X 0,Y 135.362,Z 840.191,A -85,B 0,C 180,E1 -25389.445,E2 -25389.445} C_VEL
LIN {X 0,Y 130.355,Z 842.863,A -85,B 0,C 180,E1 -25393.97,E2 -25393.97} C_VEL
LIN {X 0,Y 125.623,Z 844.678,A -85,B 0,C 180,E1 -25399.613,E2 -25399.613} C_VEL
LIN {X 0,Y 123.001,Z 845.141,A -85,B 0,C 180,E1 -25403.912,E2 -25403.912} C_VEL
LIN {X 0,Y 120.72,Z 844.808,A -85,B 0,C 180,E1 -25409.165,E2 -25409.165} C_VEL
LIN {X 0,Y 119.074,Z 842.937,A -85,B 0,C 180,E1 -25416.172,E2 -25416.172} C_VEL
LIN {X 0,Y 118.762,Z 839.651,A -85,B 0,C 180,E1 -25422.7,E2 -25422.7} C_VEL
LIN {X 0,Y 119.205,Z 836.283,A -85,B 0,C 180,E1 -25427.443,E2 -25427.443} C_VEL
LIN {X 0,Y 120.447,Z 830.716,A -85,B 0,C 180,E1 -25433.282,E2 -25433.282} C_VEL
LIN {X 0,Y 122.475,Z 823.598,A -85,B 0,C 180,E1 -25438.908,E2 -25438.908} C_VEL
LIN {X 0,Y 124.639,Z 816.629,A -85,B 0,C 180,E1 -25443.188,E2 -25443.188} C_VEL
LIN {X 0,Y 127.374,Z 808.252,A -85,B 0,C 180,E1 -25447.282,E2 -25447.282} C_VEL
LIN {X 0,Y 130.633,Z 798.141,A -85,B 0,C 180,E1 -25451.17,E2 -25451.17} C_VEL
LIN {X 0,Y 133.823,Z 787.352,A -85,B 0,C 180,E1 -25454.368,E2 -25454.368} C_VEL
LIN {X 0,Y 135.268,Z 781.884,A -85,B 0,C 180,E1 -25455.714,E2 -25455.714} C_VEL
LIN {X 0,Y 135.347,Z 771.062,A -85,B 0,C 180,E1 -25458.394,E2 -25458.394} C_VEL
LIN {X 0,Y 134.735,Z 758.546,A -85,B 0,C 180,E1 -25460.999,E2 -25460.999} C_VEL
LIN {X 0,Y 133.654,Z 746.689,A -85,B 0,C 180,E1 -25463.017,E2 -25463.017} C_VEL
LIN {X 0,Y 131.841,Z 733.388,A -85,B 0,C 180,E1 -25464.936,E2 -25464.936} C_VEL
LIN {X 0,Y 132.704,Z 730.231,A -85,B 0,C 180,E1 -25466.966,E2 -25466.966} C_VEL
LIN {X 0,Y 132.121,Z 722.122,A -85,B 0,C 180,E1 -25473.137,E2 -25473.137} C_VEL
LIN {X 0,Y 136.27,Z 726.85,A -85,B 0,C 180,E1 -25475.922,E2 -25475.922} C_VEL
LIN {X 0,Y 136.63,Z 727.627,A -85,B 0,C 180,E1 -25476.307,E2 -25476.307} C_VEL
LIN {X 0,Y 133.455,Z 737.413,A -85,B 0,C 180,E1 -25479.856,E2 -25479.856} C_VEL
LIN {X 0,Y 130.329,Z 746.221,A -85,B 0,C 180,E1 -25483.917,E2 -25483.917} C_VEL
LIN {X 0,Y 127.63,Z 753.925,A -85,B 0,C 180,E1 -25488.461,E2 -25488.461} C_VEL
LIN {X 0,Y 125.574,Z 760.09,A -85,B 0,C 180,E1 -25493.066,E2 -25493.066} C_VEL
LIN {X 0,Y 123.806,Z 766.062,A -85,B 0,C 180,E1 -25498.851,E2 -25498.851} C_VEL
LIN {X 0,Y 123.005,Z 770.508,A -85,B 0,C 180,E1 -25504.847,E2 -25504.847} C_VEL
LIN {X 0,Y 123.132,Z 772.73,A -85,B 0,C 180,E1 -25508.893,E2 -25508.893} C_VEL
LIN {X 0,Y 123.784,Z 774.297,A -85,B 0,C 180,E1 -25512.948,E2 -25512.948} C_VEL
LIN {X 0,Y 125.236,Z 775.409,A -85,B 0,C 180,E1 -25517.669,E2 -25517.669} C_VEL
LIN {X 0,Y 127.616,Z 775.681,A -85,B 0,C 180,E1 -25522.715,E2 -25522.715} C_VEL
LIN {X 0,Y 131.635,Z 774.666,A -85,B 0,C 180,E1 -25528.678,E2 -25528.678} C_VEL
LIN {X 0,Y 136.625,Z 772.176,A -85,B 0,C 180,E1 -25534.187,E2 -25534.187} C_VEL
LIN {X 0,Y 142.718,Z 768.065,A -85,B 0,C 180,E1 -25539.334,E2 -25539.334} C_VEL
LIN {X 0,Y 148.966,Z 762.875,A -85,B 0,C 180,E1 -25543.557,E2 -25543.557} C_VEL
LIN {X 0,Y 154.676,Z 757.248,A -85,B 0,C 180,E1 -25546.869,E2 -25546.869} C_VEL
LIN {X 0,Y 156.201,Z 755.634,A -85,B 0,C 180,E1 -25547.661,E2 -25547.661} C_VEL
LIN {X 0,Y 157.034,Z 754.471,A -85,B 0,C 180,E1 -25548.383,E2 -25548.383} C_VEL
LIN {X 0,Y 158.335,Z 750.056,A -85,B 0,C 180,E1 -25552.348,E2 -25552.348} C_VEL
LIN {X 0,Y 159.119,Z 745.997,A -85,B 0,C 180,E1 -25556.202,E2 -25556.202} C_VEL
LIN {X 0,Y 159.524,Z 742.46,A -85,B 0,C 180,E1 -25560,E2 -25560} C_VEL
LIN {X 0,Y 159.737,Z 740.424,A -85,B 0,C 180,E1 -25562.522,E2 -25562.522} C_VEL
LIN {X 0,Y 159.868,Z 738.697,A -85,B 0,C 180,E1 -25565.044,E2 -25565.044} C_VEL
LIN {X 0,Y 159.699,Z 737.628,A -85,B 0,C 180,E1 -25567.587,E2 -25567.587} C_VEL
LIN {X 0,Y 159.238,Z 737.391,A -85,B 0,C 180,E1 -25570.169,E2 -25570.169} C_VEL
LIN {X 0,Y 158.473,Z 738.274,A -85,B 0,C 180,E1 -25575.432,E2 -25575.432} C_VEL
LIN {X 0,Y 158.277,Z 739.288,A -85,B 0,C 180,E1 -25578.109,E2 -25578.109} C_VEL
LIN {X 0,Y 158.121,Z 740.992,A -85,B 0,C 180,E1 -25581.029,E2 -25581.029} C_VEL
LIN {X 0,Y 158.357,Z 745.072,A -85,B 0,C 180,E1 -25586.348,E2 -25586.348} C_VEL
LIN {X 0,Y 158.334,Z 748.355,A -85,B 0,C 180,E1 -25589.227,E2 -25589.227} C_VEL
LIN {X 0,Y 158.371,Z 752.109,A -85,B 0,C 180,E1 -25592.176,E2 -25592.176} C_VEL
LIN {X 0,Y 158.212,Z 756.78,A -85,B 0,C 180,E1 -25595.274,E2 -25595.274} C_VEL
LIN {X 0,Y 157.996,Z 758.128,A -85,B 0,C 180,E1 -25596.044,E2 -25596.044} C_VEL
LIN {X 0,Y 153.803,Z 767.339,A -85,B 0,C 180,E1 -25599.772,E2 -25599.772} C_VEL
LIN {X 0,Y 149.425,Z 775.28,A -85,B 0,C 180,E1 -25603.194,E2 -25603.194} C_VEL
LIN {X 0,Y 144.339,Z 783.006,A -85,B 0,C 180,E1 -25607.024,E2 -25607.024} C_VEL
LIN {X 0,Y 139.196,Z 789.536,A -85,B 0,C 180,E1 -25610.865,E2 -25610.865} C_VEL
LIN {X 0,Y 133.298,Z 796.565,A -85,B 0,C 180,E1 -25616.384,E2 -25616.384} C_VEL
LIN {X 0,Y 132.073,Z 798.11,A -85,B 0,C 180,E1 -25617.624,E2 -25617.624} C_VEL
LIN {X 0,Y 129.006,Z 808.22,A -85,B 0,C 180,E1 -25620.891,E2 -25620.891} C_VEL
LIN {X 0,Y 126.226,Z 816.885,A -85,B 0,C 180,E1 -25624.435,E2 -25624.435} C_VEL
LIN {X 0,Y 123.455,Z 825.858,A -85,B 0,C 180,E1 -25629.156,E2 -25629.156} C_VEL
LIN {X 0,Y 121.372,Z 833.059,A -85,B 0,C 180,E1 -25634.033,E2 -25634.033} C_VEL
LIN {X 0,Y 120.347,Z 837.948,A -85,B 0,C 180,E1 -25638.204,E2 -25638.204} C_VEL
LIN {X 0,Y 119.688,Z 842.644,A -85,B 0,C 180,E1 -25643.254,E2 -25643.254} C_VEL
LIN {X 0,Y 119.586,Z 845.728,A -85,B 0,C 180,E1 -25647.555,E2 -25647.555} C_VEL
LIN {X 0,Y 119.658,Z 847.138,A -85,B 0,C 180,E1 -25649.998,E2 -25649.998} C_VEL
LIN {X 0,Y 119.469,Z 848.641,A -85,B 0,C 180,E1 -25653.371,E2 -25653.371} C_VEL
LIN {X 0,Y 119.93,Z 850.501,A -85,B 0,C 180,E1 -25660.123,E2 -25660.123} C_VEL
LIN {X 0,Y 121.807,Z 850.836,A -85,B 0,C 180,E1 -25666.766,E2 -25666.766} C_VEL
LIN {X 0,Y 125.25,Z 849.738,A -85,B 0,C 180,E1 -25673.126,E2 -25673.126} C_VEL
LIN {X 0,Y 130.377,Z 847.194,A -85,B 0,C 180,E1 -25679.02,E2 -25679.02} C_VEL
LIN {X 0,Y 136.669,Z 843.092,A -85,B 0,C 180,E1 -25684.446,E2 -25684.446} C_VEL
LIN {X 0,Y 142.35,Z 838.949,A -85,B 0,C 180,E1 -25688.105,E2 -25688.105} C_VEL
LIN {X 0,Y 148.406,Z 833.804,A -85,B 0,C 180,E1 -25691.526,E2 -25691.526} C_VEL
LIN {X 0,Y 156.509,Z 826.249,A -85,B 0,C 180,E1 -25695.009,E2 -25695.009} C_VEL
LIN {X 0,Y 163.812,Z 818.275,A -85,B 0,C 180,E1 -25697.735,E2 -25697.735} C_VEL
LIN {X 0,Y 171.012,Z 808.794,A -85,B 0,C 180,E1 -25700.402,E2 -25700.402} C_VEL
LIN {X 0,Y 173.481,Z 805.107,A -85,B 0,C 180,E1 -25701.298,E2 -25701.298} C_VEL
LIN {X 0,Y 174.818,Z 802.562,A -85,B 0,C 180,E1 -25702.169,E2 -25702.169} C_VEL
LIN {X 0,Y 175.591,Z 799.897,A -85,B 0,C 180,E1 -25703.658,E2 -25703.658} C_VEL
LIN {X 0,Y 176.361,Z 796.181,A -85,B 0,C 180,E1 -25706.038,E2 -25706.038} C_VEL
LIN {X 0,Y 177.36,Z 793.756,A -85,B 0,C 180,E1 -25707.049,E2 -25707.049} C_VEL
LIN {X 0,Y 178.318,Z 791.296,A -85,B 0,C 180,E1 -25708.194,E2 -25708.194} C_VEL
LIN {X 0,Y 177.926,Z 790.193,A -85,B 0,C 180,E1 -25710.338,E2 -25710.338} C_VEL
LIN {X 0,Y 177.633,Z 789.781,A -85,B 0,C 180,E1 -25711.655,E2 -25711.655} C_VEL
LIN {X 0,Y 177.157,Z 789.587,A -85,B 0,C 180,E1 -25714.126,E2 -25714.126} C_VEL
LIN {X 0,Y 176.653,Z 790.014,A -85,B 0,C 180,E1 -25716.556,E2 -25716.556} C_VEL
LIN {X 0,Y 176.249,Z 790.994,A -85,B 0,C 180,E1 -25718.968,E2 -25718.968} C_VEL
LIN {X 0,Y 175.844,Z 792.52,A -85,B 0,C 180,E1 -25721.353,E2 -25721.353} C_VEL
LIN {X 0,Y 175.148,Z 794.85,A -85,B 0,C 180,E1 -25723.687,E2 -25723.687} C_VEL
LIN {X 0,Y 174.391,Z 796.648,A -85,B 0,C 180,E1 -25724.814,E2 -25724.814} C_VEL
LIN {X 0,Y 169.998,Z 804.509,A -85,B 0,C 180,E1 -25728.07,E2 -25728.07} C_VEL
LIN {X 0,Y 166.404,Z 809.943,A -85,B 0,C 180,E1 -25730.274,E2 -25730.274} C_VEL
LIN {X 0,Y 163.514,Z 813.451,A -85,B 0,C 180,E1 -25731.314,E2 -25731.314} C_VEL
LIN {X 0,Y 155.44,Z 821.851,A -85,B 0,C 180,E1 -25734.08,E2 -25734.08} C_VEL
LIN {X 0,Y 147.626,Z 828.806,A -85,B 0,C 180,E1 -25737.271,E2 -25737.271} C_VEL
LIN {X 0,Y 140.565,Z 834.174,A -85,B 0,C 180,E1 -25740.697,E2 -25740.697} C_VEL
LIN {X 0,Y 133.951,Z 838.484,A -85,B 0,C 180,E1 -25744.56,E2 -25744.56} C_VEL
LIN {X 0,Y 127.302,Z 842.07,A -85,B 0,C 180,E1 -25749.533,E2 -25749.533} C_VEL
LIN {X 0,Y 122.949,Z 843.912,A -85,B 0,C 180,E1 -25753.66,E2 -25753.66} C_VEL
LIN {X 0,Y 118.77,Z 845.125,A -85,B 0,C 180,E1 -25758.785,E2 -25758.785} C_VEL
LIN {X 0,Y 115.005,Z 845.276,A -85,B 0,C 180,E1 -25765.326,E2 -25765.326} C_VEL
LIN {X 0,Y 113.338,Z 844.625,A -85,B 0,C 180,E1 -25769.763,E2 -25769.763} C_VEL
LIN {X 0,Y 112.064,Z 842.965,A -85,B 0,C 180,E1 -25775.389,E2 -25775.389} C_VEL
LIN {X 0,Y 111.619,Z 840.4,A -85,B 0,C 180,E1 -25780.928,E2 -25780.928} C_VEL
LIN {X 0,Y 111.935,Z 836.937,A -85,B 0,C 180,E1 -25786.321,E2 -25786.321} C_VEL
LIN {X 0,Y 113.182,Z 831.348,A -85,B 0,C 180,E1 -25792.72,E2 -25792.72} C_VEL
LIN {X 0,Y 115.152,Z 824.411,A -85,B 0,C 180,E1 -25798.698,E2 -25798.698} C_VEL
LIN {X 0,Y 117.595,Z 816.827,A -85,B 0,C 180,E1 -25803.696,E2 -25803.696} C_VEL
LIN {X 0,Y 120.816,Z 807.28,A -85,B 0,C 180,E1 -25808.549,E2 -25808.549} C_VEL
LIN {X 0,Y 124.207,Z 797.144,A -85,B 0,C 180,E1 -25812.503,E2 -25812.503} C_VEL
LIN {X 0,Y 127.888,Z 785.097,A -85,B 0,C 180,E1 -25816.09,E2 -25816.09} C_VEL
LIN {X 0,Y 128.638,Z 781.627,A -85,B 0,C 180,E1 -25816.977,E2 -25816.977} C_VEL
LIN {X 0,Y 128.755,Z 770.515,A -85,B 0,C 180,E1 -25819.863,E2 -25819.863} C_VEL
LIN {X 0,Y 128.215,Z 757.18,A -85,B 0,C 180,E1 -25822.719,E2 -25822.719} C_VEL
LIN {X 0,Y 126.924,Z 743.903,A -85,B 0,C 180,E1 -25825.04,E2 -25825.04} C_VEL
LIN {X 0,Y 125.519,Z 733.554,A -85,B 0,C 180,E1 -25826.591,E2 -25826.591} C_VEL
LIN {X 0,Y 125.967,Z 731.983,A -85,B 0,C 180,E1 -25827.604,E2 -25827.604} C_VEL
LIN {X 0,Y 125.527,Z 725.433,A -85,B 0,C 180,E1 -25832.709,E2 -25832.709} C_VEL
LIN {X 0,Y 129.596,Z 729.882,A -85,B 0,C 180,E1 -25835.572,E2 -25835.572} C_VEL
LIN {X 0,Y 126.535,Z 738.939,A -85,B 0,C 180,E1 -25839.097,E2 -25839.097} C_VEL
LIN {X 0,Y 123.036,Z 748.414,A -85,B 0,C 180,E1 -25843.819,E2 -25843.819} C_VEL
LIN {X 0,Y 120.391,Z 755.594,A -85,B 0,C 180,E1 -25848.401,E2 -25848.401} C_VEL
LIN {X 0,Y 118.183,Z 762.071,A -85,B 0,C 180,E1 -25853.668,E2 -25853.668} C_VEL
LIN {X 0,Y 116.727,Z 766.963,A -85,B 0,C 180,E1 -25858.796,E2 -25858.796} C_VEL
LIN {X 0,Y 115.959,Z 771.46,A -85,B 0,C 180,E1 -25865.156,E2 -25865.156} C_VEL
LIN {X 0,Y 116.454,Z 774.585,A -85,B 0,C 180,E1 -25871.596,E2 -25871.596} C_VEL
LIN {X 0,Y 117.492,Z 775.915,A -85,B 0,C 180,E1 -25875.875,E2 -25875.875} C_VEL
LIN {X 0,Y 119.099,Z 776.655,A -85,B 0,C 180,E1 -25880.099,E2 -25880.099} C_VEL
LIN {X 0,Y 121.529,Z 776.75,A -85,B 0,C 180,E1 -25884.669,E2 -25884.669} C_VEL
LIN {X 0,Y 124.977,Z 775.993,A -85,B 0,C 180,E1 -25889.595,E2 -25889.595} C_VEL
LIN {X 0,Y 129.037,Z 774.339,A -85,B 0,C 180,E1 -25894.169,E2 -25894.169} C_VEL
LIN {X 0,Y 135.082,Z 770.922,A -85,B 0,C 180,E1 -25899.475,E2 -25899.475} C_VEL
LIN {X 0,Y 139.757,Z 767.632,A -85,B 0,C 180,E1 -25902.838,E2 -25902.838} C_VEL
LIN {X 0,Y 146.215,Z 762.362,A -85,B 0,C 180,E1 -25906.744,E2 -25906.744} C_VEL
LIN {X 0,Y 150.967,Z 757.838,A -85,B 0,C 180,E1 -25909.269,E2 -25909.269} C_VEL
LIN {X 0,Y 151.826,Z 756.284,A -85,B 0,C 180,E1 -25910.677,E2 -25910.677} C_VEL
LIN {X 0,Y 153.196,Z 752.293,A -85,B 0,C 180,E1 -25914.736,E2 -25914.736} C_VEL
LIN {X 0,Y 154.157,Z 748.757,A -85,B 0,C 180,E1 -25918.694,E2 -25918.694} C_VEL
LIN {X 0,Y 154.836,Z 745.748,A -85,B 0,C 180,E1 -25922.602,E2 -25922.602} C_VEL
LIN {X 0,Y 155.152,Z 744.074,A -85,B 0,C 180,E1 -25925.198,E2 -25925.198} C_VEL
LIN {X 0,Y 155.174,Z 743.108,A -85,B 0,C 180,E1 -25927.81,E2 -25927.81} C_VEL
LIN {X 0,Y 154.728,Z 743.009,A -85,B 0,C 180,E1 -25930.468,E2 -25930.468} C_VEL
LIN {X 0,Y 154.032,Z 744.112,A -85,B 0,C 180,E1 -25935.889,E2 -25935.889} C_VEL
LIN {X 0,Y 153.825,Z 745.291,A -85,B 0,C 180,E1 -25938.652,E2 -25938.652} C_VEL
LIN {X 0,Y 153.584,Z 749.065,A -85,B 0,C 180,E1 -25944.321,E2 -25944.321} C_VEL
LIN {X 0,Y 153.689,Z 750.16,A -85,B 0,C 180,E1 -25945.749,E2 -25945.749} C_VEL
LIN {X 0,Y 153.441,Z 755.059,A -85,B 0,C 180,E1 -25950.254,E2 -25950.254} C_VEL
LIN {X 0,Y 152.872,Z 760.366,A -85,B 0,C 180,E1 -25954.154,E2 -25954.154} C_VEL
LIN {X 0,Y 152.538,Z 761.536,A -85,B 0,C 180,E1 -25954.827,E2 -25954.827} C_VEL
LIN {X 0,Y 148.05,Z 769.934,A -85,B 0,C 180,E1 -25958.49,E2 -25958.49} C_VEL
LIN {X 0,Y 142.703,Z 778.148,A -85,B 0,C 180,E1 -25962.374,E2 -25962.374} C_VEL
LIN {X 0,Y 137.279,Z 785.286,A -85,B 0,C 180,E1 -25966.327,E2 -25966.327} C_VEL
LIN {X 0,Y 130.343,Z 792.911,A -85,B 0,C 180,E1 -25971.677,E2 -25971.677} C_VEL
LIN {X 0,Y 125.253,Z 798.304,A -85,B 0,C 180,E1 -25976.712,E2 -25976.712} C_VEL
LIN {X 0,Y 122.072,Z 808.431,A -85,B 0,C 180,E1 -25980.175,E2 -25980.175} C_VEL
LIN {X 0,Y 119.285,Z 816.742,A -85,B 0,C 180,E1 -25983.774,E2 -25983.774} C_VEL
LIN {X 0,Y 116.378,Z 825.692,A -85,B 0,C 180,E1 -25988.754,E2 -25988.754} C_VEL
LIN {X 0,Y 114.248,Z 832.885,A -85,B 0,C 180,E1 -25993.928,E2 -25993.928} C_VEL
LIN {X 0,Y 113.069,Z 838.638,A -85,B 0,C 180,E1 -25999.251,E2 -25999.251} C_VEL
LIN {X 0,Y 112.546,Z 843.109,A -85,B 0,C 180,E1 -26004.623,E2 -26004.623} C_VEL
LIN {X 0,Y 112.58,Z 846.446,A -85,B 0,C 180,E1 -26009.998,E2 -26009.998} C_VEL
LIN {X 0,Y 112.401,Z 848.057,A -85,B 0,C 180,E1 -26013.583,E2 -26013.583} C_VEL
LIN {X 0,Y 112.953,Z 850.088,A -85,B 0,C 180,E1 -26020.756,E2 -26020.756} C_VEL
LIN {X 0,Y 114.995,Z 850.664,A -85,B 0,C 180,E1 -26027.791,E2 -26027.791} C_VEL
LIN {X 0,Y 118.734,Z 849.763,A -85,B 0,C 180,E1 -26034.475,E2 -26034.475} C_VEL
LIN {X 0,Y 124.205,Z 847.437,A -85,B 0,C 180,E1 -26040.612,E2 -26040.612} C_VEL
LIN {X 0,Y 129.138,Z 844.724,A -85,B 0,C 180,E1 -26044.848,E2 -26044.848} C_VEL
LIN {X 0,Y 134.777,Z 841.124,A -85,B 0,C 180,E1 -26048.734,E2 -26048.734} C_VEL
LIN {X 0,Y 141.101,Z 836.533,A -85,B 0,C 180,E1 -26052.251,E2 -26052.251} C_VEL
LIN {X 0,Y 145.618,Z 832.905,A -85,B 0,C 180,E1 -26054.41,E2 -26054.41} C_VEL
LIN {X 0,Y 152.926,Z 826.447,A -85,B 0,C 180,E1 -26057.331,E2 -26057.331} C_VEL
LIN {X 0,Y 159.261,Z 820.007,A -85,B 0,C 180,E1 -26059.569,E2 -26059.569} C_VEL
LIN {X 0,Y 166.756,Z 810.992,A -85,B 0,C 180,E1 -26062.204,E2 -26062.204} C_VEL
LIN {X 0,Y 171.629,Z 804.11,A -85,B 0,C 180,E1 -26063.97,E2 -26063.97} C_VEL
LIN {X 0,Y 175.954,Z 796.574,A -85,B 0,C 180,E1 -26066.158,E2 -26066.158} C_VEL
LIN {X 0,Y 177.36,Z 793.756,A -85,B 0,C 180,E1 -26067.049,E2 -26067.049} C_VEL
LIN {X 0,Y 177.949,Z 792.28,A -85,B 0,C 180,E1 -26067.755,E2 -26067.755} C_VEL
LIN {X 0,Y 177.985,Z 791.28,A -85,B 0,C 180,E1 -26068.896,E2 -26068.896} C_VEL
LIN {X 0,Y 177.256,Z 791.207,A -85,B 0,C 180,E1 -26070.447,E2 -26070.447} C_VEL
LIN {X 0,Y 176.316,Z 791.83,A -85,B 0,C 180,E1 -26071.675,E2 -26071.675} C_VEL
LIN {X 0,Y 172.556,Z 795.875,A -85,B 0,C 180,E1 -26076.62,E2 -26076.62} C_VEL
LIN {X 0,Y 172.337,Z 796.216,A -85,B 0,C 180,E1 -26077.366,E2 -26077.366} C_VEL
LIN {X 0,Y 171.665,Z 797.667,A -85,B 0,C 180,E1 -26080.321,E2 -26080.321} C_VEL
LIN {X 0,Y 171.122,Z 799.09,A -85,B 0,C 180,E1 -26082.059,E2 -26082.059} C_VEL
LIN {X 0,Y 170.478,Z 800.51,A -85,B 0,C 180,E1 -26083.227,E2 -26083.227} C_VEL
LIN {X 0,Y 166.701,Z 806.276,A -85,B 0,C 180,E1 -26085.845,E2 -26085.845} C_VEL
LIN {X 0,Y 162.768,Z 811.741,A -85,B 0,C 180,E1 -26088.165,E2 -26088.165} C_VEL
LIN {X 0,Y 161.568,Z 813.203,A -85,B 0,C 180,E1 -26088.711,E2 -26088.711} C_VEL
LIN {X 0,Y 152.928,Z 821.795,A -85,B 0,C 180,E1 -26091.45,E2 -26091.45} C_VEL
LIN {X 0,Y 144.87,Z 828.646,A -85,B 0,C 180,E1 -26094.432,E2 -26094.432} C_VEL
LIN {X 0,Y 138.696,Z 833.153,A -85,B 0,C 180,E1 -26097.095,E2 -26097.095} C_VEL
LIN {X 0,Y 130.262,Z 838.436,A -85,B 0,C 180,E1 -26101.545,E2 -26101.545} C_VEL
LIN {X 0,Y 122.894,Z 842.134,A -85,B 0,C 180,E1 -26106.567,E2 -26106.567} C_VEL
LIN {X 0,Y 118.563,Z 843.878,A -85,B 0,C 180,E1 -26110.243,E2 -26110.243} C_VEL
LIN {X 0,Y 114.773,Z 844.984,A -85,B 0,C 180,E1 -26114.178,E2 -26114.178} C_VEL
LIN {X 0,Y 111.315,Z 845.583,A -85,B 0,C 180,E1 -26118.737,E2 -26118.737} C_VEL
LIN {X 0,Y 108.11,Z 845.403,A -85,B 0,C 180,E1 -26124.486,E2 -26124.486} C_VEL
LIN {X 0,Y 105.952,Z 844.271,A -85,B 0,C 180,E1 -26130.427,E2 -26130.427} C_VEL
LIN {X 0,Y 104.726,Z 841.89,A -85,B 0,C 180,E1 -26137.155,E2 -26137.155} C_VEL
LIN {X 0,Y 104.535,Z 839.271,A -85,B 0,C 180,E1 -26142.311,E2 -26142.311} C_VEL
LIN {X 0,Y 105.075,Z 835.402,A -85,B 0,C 180,E1 -26148.024,E2 -26148.024} C_VEL
LIN {X 0,Y 106.237,Z 830.634,A -85,B 0,C 180,E1 -26153.463,E2 -26153.463} C_VEL
LIN {X 0,Y 108.4,Z 823.35,A -85,B 0,C 180,E1 -26159.841,E2 -26159.841} C_VEL
LIN {X 0,Y 110.795,Z 816.261,A -85,B 0,C 180,E1 -26164.651,E2 -26164.651} C_VEL
LIN {X 0,Y 113.943,Z 807.342,A -85,B 0,C 180,E1 -26169.41,E2 -26169.41} C_VEL
LIN {X 0,Y 117.325,Z 797.635,A -85,B 0,C 180,E1 -26173.42,E2 -26173.42} C_VEL
LIN {X 0,Y 120.855,Z 786.554,A -85,B 0,C 180,E1 -26176.946,E2 -26176.946} C_VEL
LIN {X 0,Y 121.885,Z 783.056,A -85,B 0,C 180,E1 -26177.878,E2 -26177.878} C_VEL
LIN {X 0,Y 122.233,Z 772.085,A -85,B 0,C 180,E1 -26180.904,E2 -26180.904} C_VEL
LIN {X 0,Y 121.88,Z 759.288,A -85,B 0,C 180,E1 -26183.875,E2 -26183.875} C_VEL
LIN {X 0,Y 120.805,Z 746.07,A -85,B 0,C 180,E1 -26186.378,E2 -26186.378} C_VEL
LIN {X 0,Y 119.229,Z 733.706,A -85,B 0,C 180,E1 -26188.351,E2 -26188.351} C_VEL
LIN {X 0,Y 118.97,Z 728.862,A -85,B 0,C 180,E1 -26192.365,E2 -26192.365} C_VEL
LIN {X 0,Y 122.459,Z 732.357,A -85,B 0,C 180,E1 -26194.913,E2 -26194.913} C_VEL
LIN {X 0,Y 119.313,Z 741.197,A -85,B 0,C 180,E1 -26198.661,E2 -26198.661} C_VEL
LIN {X 0,Y 115.729,Z 750.503,A -85,B 0,C 180,E1 -26203.677,E2 -26203.677} C_VEL
LIN {X 0,Y 112.78,Z 758.214,A -85,B 0,C 180,E1 -26209.12,E2 -26209.12} C_VEL
LIN {X 0,Y 110.443,Z 765.006,A -85,B 0,C 180,E1 -26215.44,E2 -26215.44} C_VEL
LIN {X 0,Y 109.22,Z 769.541,A -85,B 0,C 180,E1 -26220.984,E2 -26220.984} C_VEL
LIN {X 0,Y 108.898,Z 772.416,A -85,B 0,C 180,E1 -26225.511,E2 -26225.511} C_VEL
LIN {X 0,Y 109.159,Z 774.688,A -85,B 0,C 180,E1 -26230.08,E2 -26230.08} C_VEL
LIN {X 0,Y 110.263,Z 776.578,A -85,B 0,C 180,E1 -26235.483,E2 -26235.483} C_VEL
LIN {X 0,Y 112.451,Z 777.712,A -85,B 0,C 180,E1 -26241.32,E2 -26241.32} C_VEL
LIN {X 0,Y 116.248,Z 777.763,A -85,B 0,C 180,E1 -26247.825,E2 -26247.825} C_VEL
LIN {X 0,Y 119.443,Z 776.996,A -85,B 0,C 180,E1 -26251.96,E2 -26251.96} C_VEL
LIN {X 0,Y 123.904,Z 775.28,A -85,B 0,C 180,E1 -26256.607,E2 -26256.607} C_VEL
LIN {X 0,Y 129.048,Z 772.627,A -85,B 0,C 180,E1 -26260.928,E2 -26260.928} C_VEL
LIN {X 0,Y 134.744,Z 768.999,A -85,B 0,C 180,E1 -26264.883,E2 -26264.883} C_VEL
LIN {X 0,Y 141.005,Z 764.267,A -85,B 0,C 180,E1 -26268.5,E2 -26268.5} C_VEL
LIN {X 0,Y 145.184,Z 760.646,A -85,B 0,C 180,E1 -26270.68,E2 -26270.68} C_VEL
LIN {X 0,Y 146.064,Z 759.462,A -85,B 0,C 180,E1 -26271.701,E2 -26271.701} C_VEL
LIN {X 0,Y 147.9,Z 755.547,A -85,B 0,C 180,E1 -26276.29,E2 -26276.29} C_VEL
LIN {X 0,Y 148.999,Z 752.641,A -85,B 0,C 180,E1 -26280,E2 -26280} C_VEL
LIN {X 0,Y 149.677,Z 750.796,A -85,B 0,C 180,E1 -26282.692,E2 -26282.692} C_VEL
LIN {X 0,Y 150.196,Z 749.221,A -85,B 0,C 180,E1 -26285.37,E2 -26285.37} C_VEL
LIN {X 0,Y 150.376,Z 748.38,A -85,B 0,C 180,E1 -26288.06,E2 -26288.06} C_VEL
LIN {X 0,Y 149.948,Z 748.408,A -85,B 0,C 180,E1 -26290.806,E2 -26290.806} C_VEL
LIN {X 0,Y 149.3,Z 749.719,A -85,B 0,C 180,E1 -26296.406,E2 -26296.406} C_VEL
LIN {X 0,Y 148.982,Z 751.179,A -85,B 0,C 180,E1 -26299.355,E2 -26299.355} C_VEL
LIN {X 0,Y 148.779,Z 755.028,A -85,B 0,C 180,E1 -26305.16,E2 -26305.16} C_VEL
LIN {X 0,Y 148.197,Z 759.514,A -85,B 0,C 180,E1 -26309.567,E2 -26309.567} C_VEL
LIN {X 0,Y 147.575,Z 763.117,A -85,B 0,C 180,E1 -26312.441,E2 -26312.441} C_VEL
LIN {X 0,Y 146.904,Z 764.932,A -85,B 0,C 180,E1 -26313.609,E2 -26313.609} C_VEL
LIN {X 0,Y 141.709,Z 773.135,A -85,B 0,C 180,E1 -26317.483,E2 -26317.483} C_VEL
LIN {X 0,Y 135.958,Z 780.71,A -85,B 0,C 180,E1 -26321.447,E2 -26321.447} C_VEL
LIN {X 0,Y 130.252,Z 787.167,A -85,B 0,C 180,E1 -26325.456,E2 -26325.456} C_VEL
LIN {X 0,Y 124.728,Z 792.57,A -85,B 0,C 180,E1 -26329.608,E2 -26329.608} C_VEL
LIN {X 0,Y 118.57,Z 798.184,A -85,B 0,C 180,E1 -26335.6,E2 -26335.6} C_VEL
LIN {X 0,Y 115.289,Z 808.112,A -85,B 0,C 180,E1 -26339.173,E2 -26339.173} C_VEL
LIN {X 0,Y 112.347,Z 816.532,A -85,B 0,C 180,E1 -26343.028,E2 -26343.028} C_VEL
LIN {X 0,Y 109.332,Z 825.451,A -85,B 0,C 180,E1 -26348.306,E2 -26348.306} C_VEL
LIN {X 0,Y 107.125,Z 832.616,A -85,B 0,C 180,E1 -26353.808,E2 -26353.808} C_VEL
LIN {X 0,Y 106.088,Z 837.489,A -85,B 0,C 180,E1 -26358.535,E2 -26358.535} C_VEL
LIN {X 0,Y 105.5,Z 842.164,A -85,B 0,C 180,E1 -26364.263,E2 -26364.263} C_VEL
LIN {X 0,Y 105.51,Z 845.688,A -85,B 0,C 180,E1 -26369.998,E2 -26369.998} C_VEL
LIN {X 0,Y 105.344,Z 847.427,A -85,B 0,C 180,E1 -26373.823,E2 -26373.823} C_VEL
LIN {X 0,Y 105.457,Z 848.746,A -85,B 0,C 180,E1 -26377.657,E2 -26377.657} C_VEL
LIN {X 0,Y 106.882,Z 850.212,A -85,B 0,C 180,E1 -26385.247,E2 -26385.247} C_VEL
LIN {X 0,Y 109.981,Z 850.271,A -85,B 0,C 180,E1 -26392.543,E2 -26392.543} C_VEL
LIN {X 0,Y 115.048,Z 848.912,A -85,B 0,C 180,E1 -26399.253,E2 -26399.253} C_VEL
LIN {X 0,Y 121.59,Z 846.091,A -85,B 0,C 180,E1 -26405.308,E2 -26405.308} C_VEL
LIN {X 0,Y 126.558,Z 843.413,A -85,B 0,C 180,E1 -26408.972,E2 -26408.972} C_VEL
LIN {X 0,Y 133.745,Z 839.001,A -85,B 0,C 180,E1 -26413.085,E2 -26413.085} C_VEL
LIN {X 0,Y 138.198,Z 835.809,A -85,B 0,C 180,E1 -26415.392,E2 -26415.392} C_VEL
LIN {X 0,Y 146.969,Z 828.968,A -85,B 0,C 180,E1 -26418.862,E2 -26418.862} C_VEL
LIN {X 0,Y 154.87,Z 821.717,A -85,B 0,C 180,E1 -26421.515,E2 -26421.515} C_VEL
LIN {X 0,Y 162.665,Z 813.163,A -85,B 0,C 180,E1 -26424.103,E2 -26424.103} C_VEL
LIN {X 0,Y 167.808,Z 806.632,A -85,B 0,C 180,E1 -26425.805,E2 -26425.805} C_VEL
LIN {X 0,Y 172.599,Z 799.217,A -85,B 0,C 180,E1 -26428.039,E2 -26428.039} C_VEL
LIN {X 0,Y 173.271,Z 798.119,A -85,B 0,C 180,E1 -26428.402,E2 -26428.402} C_VEL
LIN {X 0,Y 173.97,Z 796.323,A -85,B 0,C 180,E1 -26429.593,E2 -26429.593} C_VEL
LIN {X 0,Y 173.702,Z 795.82,A -85,B 0,C 180,E1 -26430.953,E2 -26430.953} C_VEL
LIN {X 0,Y 173.196,Z 795.466,A -85,B 0,C 180,E1 -26433.489,E2 -26433.489} C_VEL
LIN {X 0,Y 172.648,Z 795.718,A -85,B 0,C 180,E1 -26435.979,E2 -26435.979} C_VEL
LIN {X 0,Y 172.337,Z 796.216,A -85,B 0,C 180,E1 -26437.366,E2 -26437.366} C_VEL
LIN {X 0,Y 171.706,Z 797.233,A -85,B 0,C 180,E1 -26438.609,E2 -26438.609} C_VEL
LIN {X 0,Y 169.968,Z 799.74,A -85,B 0,C 180,E1 -26440.065,E2 -26440.065} C_VEL
LIN {X 0,Y 164.532,Z 807.053,A -85,B 0,C 180,E1 -26443.014,E2 -26443.014} C_VEL
LIN {X 0,Y 159.39,Z 813.442,A -85,B 0,C 180,E1 -26445.933,E2 -26445.933} C_VEL
LIN {X 0,Y 158.221,Z 814.77,A -85,B 0,C 180,E1 -26446.498,E2 -26446.498} C_VEL
LIN {X 0,Y 149.413,Z 823.05,A -85,B 0,C 180,E1 -26449.155,E2 -26449.155} C_VEL
LIN {X 0,Y 142.051,Z 828.886,A -85,B 0,C 180,E1 -26451.677,E2 -26451.677} C_VEL
LIN {X 0,Y 134.057,Z 834.317,A -85,B 0,C 180,E1 -26454.903,E2 -26454.903} C_VEL
LIN {X 0,Y 126.536,Z 838.653,A -85,B 0,C 180,E1 -26458.614,E2 -26458.614} C_VEL
LIN {X 0,Y 118.828,Z 842.231,A -85,B 0,C 180,E1 -26463.39,E2 -26463.39} C_VEL
LIN {X 0,Y 113.438,Z 844.189,A -85,B 0,C 180,E1 -26467.593,E2 -26467.593} C_VEL
LIN {X 0,Y 108.147,Z 845.506,A -85,B 0,C 180,E1 -26472.906,E2 -26472.906} C_VEL
LIN {X 0,Y 103.089,Z 845.79,A -85,B 0,C 180,E1 -26479.929,E2 -26479.929} C_VEL
LIN {X 0,Y 100.675,Z 845.256,A -85,B 0,C 180,E1 -26484.842,E2 -26484.842} C_VEL
LIN {X 0,Y 98.583,Z 843.722,A -85,B 0,C 180,E1 -26491.192,E2 -26491.192} C_VEL
LIN {X 0,Y 97.589,Z 841.261,A -85,B 0,C 180,E1 -26497.615,E2 -26497.615} C_VEL
LIN {X 0,Y 97.511,Z 837.913,A -85,B 0,C 180,E1 -26503.888,E2 -26503.888} C_VEL
LIN {X 0,Y 98.296,Z 833.652,A -85,B 0,C 180,E1 -26509.951,E2 -26509.951} C_VEL
LIN {X 0,Y 99.69,Z 828.502,A -85,B 0,C 180,E1 -26515.671,E2 -26515.671} C_VEL
LIN {X 0,Y 101.646,Z 822.366,A -85,B 0,C 180,E1 -26521.056,E2 -26521.056} C_VEL
LIN {X 0,Y 104.655,Z 813.943,A -85,B 0,C 180,E1 -26526.81,E2 -26526.81} C_VEL
LIN {X 0,Y 108.066,Z 804.574,A -85,B 0,C 180,E1 -26531.697,E2 -26531.697} C_VEL
LIN {X 0,Y 111.753,Z 794.295,A -85,B 0,C 180,E1 -26535.823,E2 -26535.823} C_VEL
LIN {X 0,Y 115.301,Z 783.287,A -85,B 0,C 180,E1 -26539.178,E2 -26539.178} C_VEL
LIN {X 0,Y 115.699,Z 773.23,A -85,B 0,C 180,E1 -26542.147,E2 -26542.147} C_VEL
LIN {X 0,Y 115.592,Z 760.975,A -85,B 0,C 180,E1 -26545.21,E2 -26545.21} C_VEL
LIN {X 0,Y 114.735,Z 747.961,A -85,B 0,C 180,E1 -26547.904,E2 -26547.904} C_VEL
LIN {X 0,Y 113.238,Z 736.225,A -85,B 0,C 180,E1 -26549.95,E2 -26549.95} C_VEL
LIN {X 0,Y 112.453,Z 733.773,A -85,B 0,C 180,E1 -26550.589,E2 -26550.589} C_VEL
LIN {X 0,Y 112.382,Z 732.218,A -85,B 0,C 180,E1 -26551.995,E2 -26551.995} C_VEL
LIN {X 0,Y 115.149,Z 734.945,A -85,B 0,C 180,E1 -26554.206,E2 -26554.206} C_VEL
LIN {X 0,Y 114.59,Z 737.255,A -85,B 0,C 180,E1 -26555.251,E2 -26555.251} C_VEL
LIN {X 0,Y 110.672,Z 746.959,A -85,B 0,C 180,E1 -26560.059,E2 -26560.059} C_VEL
LIN {X 0,Y 107.488,Z 754.887,A -85,B 0,C 180,E1 -26565.163,E2 -26565.163} C_VEL
LIN {X 0,Y 104.994,Z 761.275,A -85,B 0,C 180,E1 -26570.427,E2 -26570.427} C_VEL
LIN {X 0,Y 102.826,Z 767.65,A -85,B 0,C 180,E1 -26577.312,E2 -26577.312} C_VEL
LIN {X 0,Y 101.872,Z 772.328,A -85,B 0,C 180,E1 -26584.121,E2 -26584.121} C_VEL
LIN {X 0,Y 102.178,Z 775.66,A -85,B 0,C 180,E1 -26590.835,E2 -26590.835} C_VEL
LIN {X 0,Y 103.951,Z 777.978,A -85,B 0,C 180,E1 -26598.05,E2 -26598.05} C_VEL
LIN {X 0,Y 106.281,Z 778.864,A -85,B 0,C 180,E1 -26603.478,E2 -26603.478} C_VEL
LIN {X 0,Y 109.774,Z 778.917,A -85,B 0,C 180,E1 -26609.191,E2 -26609.191} C_VEL
LIN {X 0,Y 115.464,Z 777.594,A -85,B 0,C 180,E1 -26615.929,E2 -26615.929} C_VEL
LIN {X 0,Y 122.105,Z 774.842,A -85,B 0,C 180,E1 -26621.752,E2 -26621.752} C_VEL
LIN {X 0,Y 129.825,Z 770.432,A -85,B 0,C 180,E1 -26627.019,E2 -26627.019} C_VEL
LIN {X 0,Y 137.417,Z 765.045,A -85,B 0,C 180,E1 -26631.175,E2 -26631.175} C_VEL
LIN {X 0,Y 140.293,Z 762.61,A -85,B 0,C 180,E1 -26632.806,E2 -26632.806} C_VEL
LIN {X 0,Y 142.316,Z 759.289,A -85,B 0,C 180,E1 -26637.17,E2 -26637.17} C_VEL
LIN {X 0,Y 143.383,Z 757.332,A -85,B 0,C 180,E1 -26640,E2 -26640} C_VEL
LIN {X 0,Y 144.228,Z 755.614,A -85,B 0,C 180,E1 -26642.793,E2 -26642.793} C_VEL
LIN {X 0,Y 145.001,Z 754.149,A -85,B 0,C 180,E1 -26645.563,E2 -26645.563} C_VEL
LIN {X 0,Y 145.312,Z 753.393,A -85,B 0,C 180,E1 -26648.343,E2 -26648.343} C_VEL
LIN {X 0,Y 144.634,Z 754.069,A -85,B 0,C 180,E1 -26653.627,E2 -26653.627} C_VEL
LIN {X 0,Y 144.233,Z 755.192,A -85,B 0,C 180,E1 -26657,E2 -26657} C_VEL
LIN {X 0,Y 143.642,Z 758.614,A -85,B 0,C 180,E1 -26663.043,E2 -26663.043} C_VEL
LIN {X 0,Y 143.624,Z 759.66,A -85,B 0,C 180,E1 -26664.579,E2 -26664.579} C_VEL
LIN {X 0,Y 142.554,Z 764.506,A -85,B 0,C 180,E1 -26669.539,E2 -26669.539} C_VEL
LIN {X 0,Y 142.061,Z 766.508,A -85,B 0,C 180,E1 -26671.264,E2 -26671.264} C_VEL
LIN {X 0,Y 141.289,Z 768.033,A -85,B 0,C 180,E1 -26672.26,E2 -26672.26} C_VEL
LIN {X 0,Y 135.31,Z 776.035,A -85,B 0,C 180,E1 -26676.381,E2 -26676.381} C_VEL
LIN {X 0,Y 128.059,Z 784.196,A -85,B 0,C 180,E1 -26681.192,E2 -26681.192} C_VEL
LIN {X 0,Y 121.201,Z 790.576,A -85,B 0,C 180,E1 -26685.904,E2 -26685.904} C_VEL
LIN {X 0,Y 114.199,Z 796.454,A -85,B 0,C 180,E1 -26692.016,E2 -26692.016} C_VEL
LIN {X 0,Y 111.74,Z 798.458,A -85,B 0,C 180,E1 -26694.56,E2 -26694.56} C_VEL
LIN {X 0,Y 108.055,Z 809.033,A -85,B 0,C 180,E1 -26698.644,E2 -26698.644} C_VEL
LIN {X 0,Y 104.281,Z 819.421,A -85,B 0,C 180,E1 -26704.017,E2 -26704.017} C_VEL
LIN {X 0,Y 101.832,Z 826.479,A -85,B 0,C 180,E1 -26708.754,E2 -26708.754} C_VEL
LIN {X 0,Y 99.77,Z 833.421,A -85,B 0,C 180,E1 -26714.681,E2 -26714.681} C_VEL
LIN {X 0,Y 98.821,Z 838.105,A -85,B 0,C 180,E1 -26719.756,E2 -26719.756} C_VEL
LIN {X 0,Y 98.382,Z 842.574,A -85,B 0,C 180,E1 -26725.901,E2 -26725.901} C_VEL
LIN {X 0,Y 98.41,Z 845.418,A -85,B 0,C 180,E1 -26731.073,E2 -26731.073} C_VEL
LIN {X 0,Y 98.44,Z 848.139,A -85,B 0,C 180,E1 -26738.207,E2 -26738.207} C_VEL
LIN {X 0,Y 100.038,Z 849.868,A -85,B 0,C 180,E1 -26746.318,E2 -26746.318} C_VEL
LIN {X 0,Y 103.441,Z 850.116,A -85,B 0,C 180,E1 -26754.055,E2 -26754.055} C_VEL
LIN {X 0,Y 108.89,Z 848.994,A -85,B 0,C 180,E1 -26761.084,E2 -26761.084} C_VEL
LIN {X 0,Y 115.873,Z 846.449,A -85,B 0,C 180,E1 -26767.336,E2 -26767.336} C_VEL
LIN {X 0,Y 120.707,Z 844.164,A -85,B 0,C 180,E1 -26770.807,E2 -26770.807} C_VEL
LIN {X 0,Y 128.7,Z 839.807,A -85,B 0,C 180,E1 -26775.224,E2 -26775.224} C_VEL
LIN {X 0,Y 133.356,Z 836.784,A -85,B 0,C 180,E1 -26777.543,E2 -26777.543} C_VEL
LIN {X 0,Y 142.475,Z 830.276,A -85,B 0,C 180,E1 -26780.976,E2 -26780.976} C_VEL
LIN {X 0,Y 150.663,Z 823.4,A -85,B 0,C 180,E1 -26783.575,E2 -26783.575} C_VEL
LIN {X 0,Y 158.753,Z 815.267,A -85,B 0,C 180,E1 -26786.102,E2 -26786.102} C_VEL
LIN {X 0,Y 164.142,Z 809.057,A -85,B 0,C 180,E1 -26787.736,E2 -26787.736} C_VEL
LIN {X 0,Y 168.707,Z 802.906,A -85,B 0,C 180,E1 -26789.632,E2 -26789.632} C_VEL
LIN {X 0,Y 169.396,Z 801.805,A -85,B 0,C 180,E1 -26790.141,E2 -26790.141} C_VEL
LIN {X 0,Y 168.982,Z 801.133,A -85,B 0,C 180,E1 -26792.774,E2 -26792.774} C_VEL
LIN {X 0,Y 168.412,Z 801.255,A -85,B 0,C 180,E1 -26795.335,E2 -26795.335} C_VEL
LIN {X 0,Y 167.795,Z 801.991,A -85,B 0,C 180,E1 -26797.854,E2 -26797.854} C_VEL
LIN {X 0,Y 167.052,Z 803.27,A -85,B 0,C 180,E1 -26800.332,E2 -26800.332} C_VEL
LIN {X 0,Y 166.436,Z 804.391,A -85,B 0,C 180,E1 -26801.536,E2 -26801.536} C_VEL
LIN {X 0,Y 164.532,Z 807.053,A -85,B 0,C 180,E1 -26803.014,E2 -26803.014} C_VEL
LIN {X 0,Y 162.604,Z 809.445,A -85,B 0,C 180,E1 -26803.895,E2 -26803.895} C_VEL
LIN {X 0,Y 158.979,Z 813.328,A -85,B 0,C 180,E1 -26804.859,E2 -26804.859} C_VEL
LIN {X 0,Y 154.813,Z 817.239,A -85,B 0,C 180,E1 -26805.553,E2 -26805.553} C_VEL
LIN {X 0,Y 148.784,Z 822.255,A -85,B 0,C 180,E1 -26806.42,E2 -26806.42} C_VEL
LIN {X 0,Y 144.328,Z 825.673,A -85,B 0,C 180,E1 -26807.328,E2 -26807.328} C_VEL
LIN {X 0,Y 142.929,Z 826.733,A -85,B 0,C 180,E1 -26807.73,E2 -26807.73} C_VEL
LIN {X 0,Y 133.713,Z 833.041,A -85,B 0,C 180,E1 -26810.927,E2 -26810.927} C_VEL
LIN {X 0,Y 123.962,Z 838.498,A -85,B 0,C 180,E1 -26815.121,E2 -26815.121} C_VEL
LIN {X 0,Y 115.162,Z 842.347,A -85,B 0,C 180,E1 -26819.999,E2 -26819.999} C_VEL
LIN {X 0,Y 109.913,Z 844.136,A -85,B 0,C 180,E1 -26823.666,E2 -26823.666} C_VEL
LIN {X 0,Y 105.187,Z 845.336,A -85,B 0,C 180,E1 -26827.679,E2 -26827.679} C_VEL
LIN {X 0,Y 100.745,Z 846.008,A -85,B 0,C 180,E1 -26832.418,E2 -26832.418} C_VEL
LIN {X 0,Y 96.393,Z 845.932,A -85,B 0,C 180,E1 -26838.597,E2 -26838.597} C_VEL
LIN {X 0,Y 92.556,Z 844.468,A -85,B 0,C 180,E1 -26847.103,E2 -26847.103} C_VEL
LIN {X 0,Y 90.689,Z 841.67,A -85,B 0,C 180,E1 -26855.535,E2 -26855.535} C_VEL
LIN {X 0,Y 90.353,Z 838.842,A -85,B 0,C 180,E1 -26861.505,E2 -26861.505} C_VEL
LIN {X 0,Y 90.856,Z 834.946,A -85,B 0,C 180,E1 -26867.852,E2 -26867.852} C_VEL
LIN {X 0,Y 92.214,Z 829.655,A -85,B 0,C 180,E1 -26874.506,E2 -26874.506} C_VEL
LIN {X 0,Y 94.627,Z 822.156,A -85,B 0,C 180,E1 -26881.709,E2 -26881.709} C_VEL
LIN {X 0,Y 97.658,Z 814.054,A -85,B 0,C 180,E1 -26887.598,E2 -26887.598} C_VEL
LIN {X 0,Y 101.288,Z 804.588,A -85,B 0,C 180,E1 -26892.851,E2 -26892.851} C_VEL
LIN {X 0,Y 104.883,Z 795.018,A -85,B 0,C 180,E1 -26896.932,E2 -26896.932} C_VEL
LIN {X 0,Y 108.301,Z 785.099,A -85,B 0,C 180,E1 -26900.194,E2 -26900.194} C_VEL
LIN {X 0,Y 108.889,Z 781.884,A -85,B 0,C 180,E1 -26901.185,E2 -26901.185} C_VEL
LIN {X 0,Y 109.303,Z 771.145,A -85,B 0,C 180,E1 -26904.467,E2 -26904.467} C_VEL
LIN {X 0,Y 109.243,Z 758.752,A -85,B 0,C 180,E1 -26907.584,E2 -26907.584} C_VEL
LIN {X 0,Y 108.299,Z 745.335,A -85,B 0,C 180,E1 -26910.424,E2 -26910.424} C_VEL
LIN {X 0,Y 107.428,Z 738.857,A -85,B 0,C 180,E1 -26911.651,E2 -26911.651} C_VEL
LIN {X 0,Y 106.508,Z 736.326,A -85,B 0,C 180,E1 -26912.363,E2 -26912.363} C_VEL
LIN {X 0,Y 108.151,Z 737.87,A -85,B 0,C 180,E1 -26913.728,E2 -26913.728} C_VEL
LIN {X 0,Y 104.027,Z 747.57,A -85,B 0,C 180,E1 -26918.745,E2 -26918.745} C_VEL
LIN {X 0,Y 100.341,Z 756.285,A -85,B 0,C 180,E1 -26924.699,E2 -26924.699} C_VEL
LIN {X 0,Y 97.511,Z 763.356,A -85,B 0,C 180,E1 -26931.125,E2 -26931.125} C_VEL
LIN {X 0,Y 95.564,Z 769.157,A -85,B 0,C 180,E1 -26938.055,E2 -26938.055} C_VEL
LIN {X 0,Y 94.784,Z 774.267,A -85,B 0,C 180,E1 -26946.385,E2 -26946.385} C_VEL
LIN {X 0,Y 95.37,Z 776.962,A -85,B 0,C 180,E1 -26952.531,E2 -26952.531} C_VEL
LIN {X 0,Y 97.253,Z 779.015,A -85,B 0,C 180,E1 -26959.43,E2 -26959.43} C_VEL
LIN {X 0,Y 100.783,Z 780.044,A -85,B 0,C 180,E1 -26966.807,E2 -26966.807} C_VEL
LIN {X 0,Y 104.231,Z 780.002,A -85,B 0,C 180,E1 -26971.837,E2 -26971.837} C_VEL
LIN {X 0,Y 108.99,Z 779.066,A -85,B 0,C 180,E1 -26977.239,E2 -26977.239} C_VEL
LIN {X 0,Y 114.442,Z 777.215,A -85,B 0,C 180,E1 -26982.119,E2 -26982.119} C_VEL
LIN {X 0,Y 122.309,Z 773.491,A -85,B 0,C 180,E1 -26987.65,E2 -26987.65} C_VEL
LIN {X 0,Y 129.6,Z 769.084,A -85,B 0,C 180,E1 -26991.724,E2 -26991.724} C_VEL
LIN {X 0,Y 134.268,Z 765.793,A -85,B 0,C 180,E1 -26994.007,E2 -26994.007} C_VEL
LIN {X 0,Y 135.231,Z 764.755,A -85,B 0,C 180,E1 -26995.287,E2 -26995.287} C_VEL
LIN {X 0,Y 137.445,Z 761.782,A -85,B 0,C 180,E1 -27000,E2 -27000} C_VEL
LIN {X 0,Y 138.558,Z 760.167,A -85,B 0,C 180,E1 -27002.908,E2 -27002.908} C_VEL
LIN {X 0,Y 139.579,Z 758.824,A -85,B 0,C 180,E1 -27005.78,E2 -27005.78} C_VEL
LIN {X 0,Y 139.978,Z 758.174,A -85,B 0,C 180,E1 -27008.663,E2 -27008.663} C_VEL
LIN {X 0,Y 139.63,Z 758.528,A -85,B 0,C 180,E1 -27011.615,E2 -27011.615} C_VEL
LIN {X 0,Y 139.067,Z 759.804,A -85,B 0,C 180,E1 -27016.216,E2 -27016.216} C_VEL
LIN {X 0,Y 138.453,Z 762.096,A -85,B 0,C 180,E1 -27020.814,E2 -27020.814} C_VEL
LIN {X 0,Y 138.172,Z 764.05,A -85,B 0,C 180,E1 -27024.012,E2 -27024.012} C_VEL
LIN {X 0,Y 136.761,Z 768.74,A -85,B 0,C 180,E1 -27029.116,E2 -27029.116} C_VEL
LIN {X 0,Y 136.368,Z 769.816,A -85,B 0,C 180,E1 -27030.116,E2 -27030.116} C_VEL
LIN {X 0,Y 134.564,Z 772.21,A -85,B 0,C 180,E1 -27031.486,E2 -27031.486} C_VEL
LIN {X 0,Y 128.895,Z 778.633,A -85,B 0,C 180,E1 -27035.125,E2 -27035.125} C_VEL
LIN {X 0,Y 122.11,Z 785.278,A -85,B 0,C 180,E1 -27039.453,E2 -27039.453} C_VEL
LIN {X 0,Y 114.095,Z 791.844,A -85,B 0,C 180,E1 -27044.895,E2 -27044.895} C_VEL
LIN {X 0,Y 106.871,Z 797.074,A -85,B 0,C 180,E1 -27051.335,E2 -27051.335} C_VEL
LIN {X 0,Y 105.028,Z 798.465,A -85,B 0,C 180,E1 -27053.29,E2 -27053.29} C_VEL
LIN {X 0,Y 101.307,Z 808.724,A -85,B 0,C 180,E1 -27057.474,E2 -27057.474} C_VEL
LIN {X 0,Y 97.935,Z 817.542,A -85,B 0,C 180,E1 -27062.193,E2 -27062.193} C_VEL
LIN {X 0,Y 94.798,Z 826.158,A -85,B 0,C 180,E1 -27068.24,E2 -27068.24} C_VEL
LIN {X 0,Y 92.677,Z 833.094,A -85,B 0,C 180,E1 -27074.606,E2 -27074.606} C_VEL
LIN {X 0,Y 91.602,Z 838.603,A -85,B 0,C 180,E1 -27081.171,E2 -27081.171} C_VEL
LIN {X 0,Y 91.379,Z 843.528,A -85,B 0,C 180,E1 -27089.007,E2 -27089.007} C_VEL
LIN {X 0,Y 91.246,Z 846.009,A -85,B 0,C 180,E1 -27094.415,E2 -27094.415} C_VEL
LIN {X 0,Y 92.102,Z 848.654,A -85,B 0,C 180,E1 -27103.231,E2 -27103.231} C_VEL
LIN {X 0,Y 94.844,Z 849.866,A -85,B 0,C 180,E1 -27111.744,E2 -27111.744} C_VEL
LIN {X 0,Y 99.709,Z 849.674,A -85,B 0,C 180,E1 -27119.561,E2 -27119.561} C_VEL
LIN {X 0,Y 106.413,Z 848.079,A -85,B 0,C 180,E1 -27126.467,E2 -27126.467} C_VEL
LIN {X 0,Y 114.887,Z 844.915,A -85,B 0,C 180,E1 -27132.77,E2 -27132.77} C_VEL
LIN {X 0,Y 123.829,Z 840.569,A -85,B 0,C 180,E1 -27137.543,E2 -27137.543} C_VEL
LIN {X 0,Y 128.716,Z 837.736,A -85,B 0,C 180,E1 -27139.851,E2 -27139.851} C_VEL
LIN {X 0,Y 136.797,Z 832.549,A -85,B 0,C 180,E1 -27142.777,E2 -27142.777} C_VEL
LIN {X 0,Y 146.653,Z 825.06,A -85,B 0,C 180,E1 -27145.754,E2 -27145.754} C_VEL
LIN {X 0,Y 156.474,Z 815.936,A -85,B 0,C 180,E1 -27148.578,E2 -27148.578} C_VEL
LIN {X 0,Y 161.98,Z 809.961,A -85,B 0,C 180,E1 -27150.196,E2 -27150.196} C_VEL
LIN {X 0,Y 164.079,Z 807.371,A -85,B 0,C 180,E1 -27151.017,E2 -27151.017} C_VEL
LIN {X 0,Y 164.455,Z 806.625,A -85,B 0,C 180,E1 -27151.96,E2 -27151.96} C_VEL
LIN {X 0,Y 163.884,Z 806.578,A -85,B 0,C 180,E1 -27154.606,E2 -27154.606} C_VEL
LIN {X 0,Y 163.187,Z 807.135,A -85,B 0,C 180,E1 -27157.194,E2 -27157.194} C_VEL
LIN {X 0,Y 162.323,Z 808.334,A -85,B 0,C 180,E1 -27159.734,E2 -27159.734} C_VEL
LIN {X 0,Y 161.245,Z 809.696,A -85,B 0,C 180,E1 -27160.919,E2 -27160.919} C_VEL
LIN {X 0,Y 157.302,Z 814.149,A -85,B 0,C 180,E1 -27163.117,E2 -27163.117} C_VEL
LIN {X 0,Y 155.024,Z 816.56,A -85,B 0,C 180,E1 -27164.216,E2 -27164.216} C_VEL
LIN {X 0,Y 147.323,Z 823.306,A -85,B 0,C 180,E1 -27166.416,E2 -27166.416} C_VEL
LIN {X 0,Y 142.929,Z 826.733,A -85,B 0,C 180,E1 -27167.73,E2 -27167.73} C_VEL
LIN {X 0,Y 138.588,Z 829.755,A -85,B 0,C 180,E1 -27168.813,E2 -27168.813} C_VEL
LIN {X 0,Y 130.42,Z 834.425,A -85,B 0,C 180,E1 -27170.172,E2 -27170.172} C_VEL
LIN {X 0,Y 122.122,Z 838.368,A -85,B 0,C 180,E1 -27171.823,E2 -27171.823} C_VEL
LIN {X 0,Y 117.67,Z 840.252,A -85,B 0,C 180,E1 -27173.421,E2 -27173.421} C_VEL
LIN {X 0,Y 111.972,Z 842.489,A -85,B 0,C 180,E1 -27176.401,E2 -27176.401} C_VEL
LIN {X 0,Y 105.42,Z 844.518,A -85,B 0,C 180,E1 -27180.558,E2 -27180.558} C_VEL
LIN {X 0,Y 98.904,Z 845.885,A -85,B 0,C 180,E1 -27185.857,E2 -27185.857} C_VEL
LIN {X 0,Y 92.306,Z 846.297,A -85,B 0,C 180,E1 -27193.203,E2 -27193.203} C_VEL
LIN {X 0,Y 88.934,Z 845.818,A -85,B 0,C 180,E1 -27198.514,E2 -27198.514} C_VEL
LIN {X 0,Y 85.773,Z 844.391,A -85,B 0,C 180,E1 -27205.676,E2 -27205.676} C_VEL
LIN {X 0,Y 83.913,Z 842.038,A -85,B 0,C 180,E1 -27213.125,E2 -27213.125} C_VEL
LIN {X 0,Y 83.288,Z 838.774,A -85,B 0,C 180,E1 -27220.59,E2 -27220.59} C_VEL
LIN {X 0,Y 83.907,Z 833.884,A -85,B 0,C 180,E1 -27228.923,E2 -27228.923} C_VEL
LIN {X 0,Y 85.299,Z 828.829,A -85,B 0,C 180,E1 -27235.479,E2 -27235.479} C_VEL
LIN {X 0,Y 87.494,Z 822.34,A -85,B 0,C 180,E1 -27242.076,E2 -27242.076} C_VEL
LIN {X 0,Y 90.658,Z 814.14,A -85,B 0,C 180,E1 -27248.474,E2 -27248.474} C_VEL
LIN {X 0,Y 94.144,Z 805.486,A -85,B 0,C 180,E1 -27253.637,E2 -27253.637} C_VEL
LIN {X 0,Y 98.092,Z 795.484,A -85,B 0,C 180,E1 -27258.211,E2 -27258.211} C_VEL
LIN {X 0,Y 102.101,Z 784.212,A -85,B 0,C 180,E1 -27262.089,E2 -27262.089} C_VEL
LIN {X 0,Y 102.782,Z 775.245,A -85,B 0,C 180,E1 -27265.099,E2 -27265.099} C_VEL
LIN {X 0,Y 103.089,Z 761.608,A -85,B 0,C 180,E1 -27268.943,E2 -27268.943} C_VEL
LIN {X 0,Y 102.448,Z 747.989,A -85,B 0,C 180,E1 -27272.131,E2 -27272.131} C_VEL
LIN {X 0,Y 102.167,Z 744.512,A -85,B 0,C 180,E1 -27272.86,E2 -27272.86} C_VEL
LIN {X 0,Y 100.274,Z 743.221,A -85,B 0,C 180,E1 -27273.844,E2 -27273.844} C_VEL
LIN {X 0,Y 99.945,Z 742.674,A -85,B 0,C 180,E1 -27274.12,E2 -27274.12} C_VEL
LIN {X 0,Y 95.97,Z 751.548,A -85,B 0,C 180,E1 -27279.486,E2 -27279.486} C_VEL
LIN {X 0,Y 92.588,Z 759.055,A -85,B 0,C 180,E1 -27285.407,E2 -27285.407} C_VEL
LIN {X 0,Y 90.3,Z 764.562,A -85,B 0,C 180,E1 -27290.942,E2 -27290.942} C_VEL
LIN {X 0,Y 88.263,Z 770.612,A -85,B 0,C 180,E1 -27298.852,E2 -27298.852} C_VEL
LIN {X 0,Y 87.741,Z 775.089,A -85,B 0,C 180,E1 -27306.775,E2 -27306.775} C_VEL
LIN {X 0,Y 88.876,Z 778.489,A -85,B 0,C 180,E1 -27315.375,E2 -27315.375} C_VEL
LIN {X 0,Y 90.974,Z 780.196,A -85,B 0,C 180,E1 -27321.829,E2 -27321.829} C_VEL
LIN {X 0,Y 94.416,Z 781.126,A -85,B 0,C 180,E1 -27328.597,E2 -27328.597} C_VEL
LIN {X 0,Y 99.99,Z 780.92,A -85,B 0,C 180,E1 -27336.031,E2 -27336.031} C_VEL
LIN {X 0,Y 104.389,Z 780.047,A -85,B 0,C 180,E1 -27340.489,E2 -27340.489} C_VEL
LIN {X 0,Y 110.159,Z 778.219,A -85,B 0,C 180,E1 -27345.215,E2 -27345.215} C_VEL
LIN {X 0,Y 118.413,Z 774.533,A -85,B 0,C 180,E1 -27350.566,E2 -27350.566} C_VEL
LIN {X 0,Y 126.995,Z 769.584,A -85,B 0,C 180,E1 -27354.975,E2 -27354.975} C_VEL
LIN {X 0,Y 129.653,Z 767.645,A -85,B 0,C 180,E1 -27356.893,E2 -27356.893} C_VEL
LIN {X 0,Y 131.268,Z 765.96,A -85,B 0,C 180,E1 -27360,E2 -27360} C_VEL
LIN {X 0,Y 132.659,Z 764.462,A -85,B 0,C 180,E1 -27363.037,E2 -27363.037} C_VEL
LIN {X 0,Y 133.936,Z 763.235,A -85,B 0,C 180,E1 -27366.024,E2 -27366.024} C_VEL
LIN {X 0,Y 134.416,Z 762.705,A -85,B 0,C 180,E1 -27369.025,E2 -27369.025} C_VEL
LIN {X 0,Y 134.037,Z 763.221,A -85,B 0,C 180,E1 -27372.107,E2 -27372.107} C_VEL
LIN {X 0,Y 133.683,Z 764.058,A -85,B 0,C 180,E1 -27375.24,E2 -27375.24} C_VEL
LIN {X 0,Y 133.148,Z 765.455,A -85,B 0,C 180,E1 -27378.464,E2 -27378.464} C_VEL
LIN {X 0,Y 132.419,Z 768.372,A -85,B 0,C 180,E1 -27383.693,E2 -27383.693} C_VEL
LIN {X 0,Y 131.019,Z 772.015,A -85,B 0,C 180,E1 -27387.993,E2 -27387.993} C_VEL
LIN {X 0,Y 130.145,Z 773.305,A -85,B 0,C 180,E1 -27389.079,E2 -27389.079} C_VEL
LIN {X 0,Y 124.806,Z 778.817,A -85,B 0,C 180,E1 -27392.361,E2 -27392.361} C_VEL
LIN {X 0,Y 117.606,Z 785.183,A -85,B 0,C 180,E1 -27396.698,E2 -27396.698} C_VEL
LIN {X 0,Y 111.286,Z 789.955,A -85,B 0,C 180,E1 -27400.724,E2 -27400.724} C_VEL
LIN {X 0,Y 103.181,Z 795.386,A -85,B 0,C 180,E1 -27407.065,E2 -27407.065} C_VEL
LIN {X 0,Y 98.427,Z 798.226,A -85,B 0,C 180,E1 -27411.808,E2 -27411.808} C_VEL
LIN {X 0,Y 94.598,Z 808.262,A -85,B 0,C 180,E1 -27416.135,E2 -27416.135} C_VEL
LIN {X 0,Y 91.068,Z 817.099,A -85,B 0,C 180,E1 -27421.16,E2 -27421.16} C_VEL
LIN {X 0,Y 87.757,Z 825.744,A -85,B 0,C 180,E1 -27427.639,E2 -27427.639} C_VEL
LIN {X 0,Y 85.574,Z 832.722,A -85,B 0,C 180,E1 -27434.517,E2 -27434.517} C_VEL
LIN {X 0,Y 84.625,Z 837.417,A -85,B 0,C 180,E1 -27440.436,E2 -27440.436} C_VEL
LIN {X 0,Y 84.282,Z 841.916,A -85,B 0,C 180,E1 -27447.61,E2 -27447.61} C_VEL
LIN {X 0,Y 84.352,Z 843.654,A -85,B 0,C 180,E1 -27451.071,E2 -27451.071} C_VEL
LIN {X 0,Y 84.471,Z 846.845,A -85,B 0,C 180,E1 -27459.576,E2 -27459.576} C_VEL
LIN {X 0,Y 86.494,Z 848.981,A -85,B 0,C 180,E1 -27468.964,E2 -27468.964} C_VEL
LIN {X 0,Y 90.638,Z 849.706,A -85,B 0,C 180,E1 -27477.723,E2 -27477.723} C_VEL
LIN {X 0,Y 96.972,Z 849.09,A -85,B 0,C 180,E1 -27485.433,E2 -27485.433} C_VEL
LIN {X 0,Y 104.936,Z 847.047,A -85,B 0,C 180,E1 -27492.044,E2 -27492.044} C_VEL
LIN {X 0,Y 109.328,Z 845.515,A -85,B 0,C 180,E1 -27494.998,E2 -27494.998} C_VEL
LIN {X 0,Y 119.185,Z 841.339,A -85,B 0,C 180,E1 -27500.044,E2 -27500.044} C_VEL
LIN {X 0,Y 124.301,Z 838.665,A -85,B 0,C 180,E1 -27502.328,E2 -27502.328} C_VEL
LIN {X 0,Y 135.555,Z 831.907,A -85,B 0,C 180,E1 -27506.048,E2 -27506.048} C_VEL
LIN {X 0,Y 144.32,Z 825.553,A -85,B 0,C 180,E1 -27508.449,E2 -27508.449} C_VEL
LIN {X 0,Y 154.5,Z 816.615,A -85,B 0,C 180,E1 -27511.119,E2 -27511.119} C_VEL
LIN {X 0,Y 158.77,Z 812.346,A -85,B 0,C 180,E1 -27512.285,E2 -27512.285} C_VEL
LIN {X 0,Y 159.106,Z 811.662,A -85,B 0,C 180,E1 -27513.786,E2 -27513.786} C_VEL
LIN {X 0,Y 158.354,Z 812.05,A -85,B 0,C 180,E1 -27516.457,E2 -27516.457} C_VEL
LIN {X 0,Y 157.293,Z 813.235,A -85,B 0,C 180,E1 -27519.056,E2 -27519.056} C_VEL
LIN {X 0,Y 155.5,Z 814.999,A -85,B 0,C 180,E1 -27520.185,E2 -27520.185} C_VEL
LIN {X 0,Y 152.036,Z 818.299,A -85,B 0,C 180,E1 -27521.818,E2 -27521.818} C_VEL
LIN {X 0,Y 148.703,Z 821.204,A -85,B 0,C 180,E1 -27522.819,E2 -27522.819} C_VEL
LIN {X 0,Y 139.19,Z 828.368,A -85,B 0,C 180,E1 -27525.376,E2 -27525.376} C_VEL
LIN {X 0,Y 129.001,Z 834.71,A -85,B 0,C 180,E1 -27528.698,E2 -27528.698} C_VEL
LIN {X 0,Y 120.63,Z 838.979,A -85,B 0,C 180,E1 -27532.054,E2 -27532.054} C_VEL
LIN {X 0,Y 117.67,Z 840.252,A -85,B 0,C 180,E1 -27533.421,E2 -27533.421} C_VEL
LIN {X 0,Y 113.246,Z 841.94,A -85,B 0,C 180,E1 -27535.195,E2 -27535.195} C_VEL
LIN {X 0,Y 104.96,Z 844.265,A -85,B 0,C 180,E1 -27537.799,E2 -27537.799} C_VEL
LIN {X 0,Y 96.906,Z 845.829,A -85,B 0,C 180,E1 -27540.92,E2 -27540.92} C_VEL
LIN {X 0,Y 92.986,Z 846.275,A -85,B 0,C 180,E1 -27543.543,E2 -27543.543} C_VEL
LIN {X 0,Y 85.961,Z 846.436,A -85,B 0,C 180,E1 -27551.174,E2 -27551.174} C_VEL
LIN {X 0,Y 80.492,Z 845.13,A -85,B 0,C 180,E1 -27560.441,E2 -27560.441} C_VEL
LIN {X 0,Y 77.366,Z 842.507,A -85,B 0,C 180,E1 -27569.974,E2 -27569.974} C_VEL
LIN {X 0,Y 76.213,Z 838.368,A -85,B 0,C 180,E1 -27580.202,E2 -27580.202} C_VEL
LIN {X 0,Y 76.587,Z 834.549,A -85,B 0,C 180,E1 -27587.232,E2 -27587.232} C_VEL
LIN {X 0,Y 78.244,Z 828.429,A -85,B 0,C 180,E1 -27595.979,E2 -27595.979} C_VEL
LIN {X 0,Y 80.524,Z 822.047,A -85,B 0,C 180,E1 -27602.928,E2 -27602.928} C_VEL
LIN {X 0,Y 83.688,Z 814.219,A -85,B 0,C 180,E1 -27609.487,E2 -27609.487} C_VEL
LIN {X 0,Y 87.569,Z 805.069,A -85,B 0,C 180,E1 -27615.284,E2 -27615.284} C_VEL
LIN {X 0,Y 91.653,Z 795.234,A -85,B 0,C 180,E1 -27619.981,E2 -27619.981} C_VEL
LIN {X 0,Y 95.497,Z 785.034,A -85,B 0,C 180,E1 -27623.664,E2 -27623.664} C_VEL
LIN {X 0,Y 96.296,Z 779,A -85,B 0,C 180,E1 -27625.817,E2 -27625.817} C_VEL
LIN {X 0,Y 96.909,Z 766.04,A -85,B 0,C 180,E1 -27630.002,E2 -27630.002} C_VEL
LIN {X 0,Y 96.81,Z 754.354,A -85,B 0,C 180,E1 -27633.123,E2 -27633.123} C_VEL
LIN {X 0,Y 96.739,Z 752.134,A -85,B 0,C 180,E1 -27633.647,E2 -27633.647} C_VEL
LIN {X 0,Y 95.134,Z 752.548,A -85,B 0,C 180,E1 -27634.239,E2 -27634.239} C_VEL
LIN {X 0,Y 91.574,Z 752.564,A -85,B 0,C 180,E1 -27635.862,E2 -27635.862} C_VEL
LIN {X 0,Y 90.094,Z 751.369,A -85,B 0,C 180,E1 -27636.886,E2 -27636.886} C_VEL
LIN {X 0,Y 89.83,Z 751.121,A -85,B 0,C 180,E1 -27637.185,E2 -27637.185} C_VEL
LIN {X 0,Y 86.474,Z 758.141,A -85,B 0,C 180,E1 -27642.769,E2 -27642.769} C_VEL
LIN {X 0,Y 83.482,Z 764.85,A -85,B 0,C 180,E1 -27649.681,E2 -27649.681} C_VEL
LIN {X 0,Y 81.355,Z 770.679,A -85,B 0,C 180,E1 -27657.627,E2 -27657.627} C_VEL
LIN {X 0,Y 80.706,Z 776.029,A -85,B 0,C 180,E1 -27667.562,E2 -27667.562} C_VEL
LIN {X 0,Y 82.06,Z 779.459,A -85,B 0,C 180,E1 -27676.753,E2 -27676.753} C_VEL
LIN {X 0,Y 85.289,Z 781.531,A -85,B 0,C 180,E1 -27685.493,E2 -27685.493} C_VEL
LIN {X 0,Y 88.818,Z 782.249,A -85,B 0,C 180,E1 -27691.656,E2 -27691.656} C_VEL
LIN {X 0,Y 93.854,Z 782.155,A -85,B 0,C 180,E1 -27698.013,E2 -27698.013} C_VEL
LIN {X 0,Y 101.735,Z 780.609,A -85,B 0,C 180,E1 -27705.278,E2 -27705.278} C_VEL
LIN {X 0,Y 110.265,Z 777.659,A -85,B 0,C 180,E1 -27711.097,E2 -27711.097} C_VEL
LIN {X 0,Y 119.759,Z 773.093,A -85,B 0,C 180,E1 -27716.08,E2 -27716.08} C_VEL
LIN {X 0,Y 121.053,Z 772.395,A -85,B 0,C 180,E1 -27716.672,E2 -27716.672} C_VEL
LIN {X 0,Y 123.928,Z 770.626,A -85,B 0,C 180,E1 -27718.376,E2 -27718.376} C_VEL
LIN {X 0,Y 126.748,Z 768.342,A -85,B 0,C 180,E1 -27723.537,E2 -27723.537} C_VEL
LIN {X 0,Y 128.061,Z 767.354,A -85,B 0,C 180,E1 -27726.302,E2 -27726.302} C_VEL
LIN {X 0,Y 128.602,Z 767.002,A -85,B 0,C 180,E1 -27729.437,E2 -27729.437} C_VEL
LIN {X 0,Y 128.213,Z 767.647,A -85,B 0,C 180,E1 -27732.666,E2 -27732.666} C_VEL
LIN {X 0,Y 127.73,Z 768.665,A -85,B 0,C 180,E1 -27735.969,E2 -27735.969} C_VEL
LIN {X 0,Y 127.07,Z 770.443,A -85,B 0,C 180,E1 -27739.905,E2 -27739.905} C_VEL
LIN {X 0,Y 126.604,Z 772.027,A -85,B 0,C 180,E1 -27742.867,E2 -27742.867} C_VEL
LIN {X 0,Y 125.23,Z 774.933,A -85,B 0,C 180,E1 -27746.678,E2 -27746.678} C_VEL
LIN {X 0,Y 122.212,Z 777.895,A -85,B 0,C 180,E1 -27748.718,E2 -27748.718} C_VEL
LIN {X 0,Y 113.857,Z 784.707,A -85,B 0,C 180,E1 -27753.453,E2 -27753.453} C_VEL
LIN {X 0,Y 106.712,Z 789.672,A -85,B 0,C 180,E1 -27757.783,E2 -27757.783} C_VEL
LIN {X 0,Y 97.998,Z 794.791,A -85,B 0,C 180,E1 -27764.177,E2 -27764.177} C_VEL
LIN {X 0,Y 91.826,Z 798.102,A -85,B 0,C 180,E1 -27770.201,E2 -27770.201} C_VEL
LIN {X 0,Y 87.962,Z 807.757,A -85,B 0,C 180,E1 -27774.599,E2 -27774.599} C_VEL
LIN {X 0,Y 84.217,Z 816.65,A -85,B 0,C 180,E1 -27779.951,E2 -27779.951} C_VEL
LIN {X 0,Y 80.747,Z 825.336,A -85,B 0,C 180,E1 -27786.939,E2 -27786.939} C_VEL
LIN {X 0,Y 78.471,Z 832.315,A -85,B 0,C 180,E1 -27794.411,E2 -27794.411} C_VEL
LIN {X 0,Y 77.397,Z 837.871,A -85,B 0,C 180,E1 -27802.169,E2 -27802.169} C_VEL
LIN {X 0,Y 77.329,Z 842.179,A -85,B 0,C 180,E1 -27809.997,E2 -27809.997} C_VEL
LIN {X 0,Y 77.212,Z 844.344,A -85,B 0,C 180,E1 -27815.22,E2 -27815.22} C_VEL
LIN {X 0,Y 78.335,Z 847.467,A -85,B 0,C 180,E1 -27825.611,E2 -27825.611} C_VEL
LIN {X 0,Y 81.772,Z 849.141,A -85,B 0,C 180,E1 -27835.447,E2 -27835.447} C_VEL
LIN {X 0,Y 87.632,Z 849.419,A -85,B 0,C 180,E1 -27844.149,E2 -27844.149} C_VEL
LIN {X 0,Y 95.372,Z 848.351,A -85,B 0,C 180,E1 -27851.542,E2 -27851.542} C_VEL
LIN {X 0,Y 104.45,Z 845.939,A -85,B 0,C 180,E1 -27857.74,E2 -27857.74} C_VEL
LIN {X 0,Y 114.79,Z 842.026,A -85,B 0,C 180,E1 -27862.739,E2 -27862.739} C_VEL
LIN {X 0,Y 120.135,Z 839.547,A -85,B 0,C 180,E1 -27864.982,E2 -27864.982} C_VEL
LIN {X 0,Y 128.834,Z 834.948,A -85,B 0,C 180,E1 -27867.726,E2 -27867.726} C_VEL
LIN {X 0,Y 139.332,Z 828.241,A -85,B 0,C 180,E1 -27870.467,E2 -27870.467} C_VEL
LIN {X 0,Y 149.809,Z 820.089,A -85,B 0,C 180,E1 -27873.039,E2 -27873.039} C_VEL
LIN {X 0,Y 152.663,Z 817.621,A -85,B 0,C 180,E1 -27873.676,E2 -27873.676} C_VEL
LIN {X 0,Y 153.299,Z 816.765,A -85,B 0,C 180,E1 -27875.631,E2 -27875.631} C_VEL
LIN {X 0,Y 152.755,Z 817.196,A -85,B 0,C 180,E1 -27876.945,E2 -27876.945} C_VEL
LIN {X 0,Y 151.699,Z 818.116,A -85,B 0,C 180,E1 -27878.245,E2 -27878.245} C_VEL
LIN {X 0,Y 147.95,Z 821.268,A -85,B 0,C 180,E1 -27879.854,E2 -27879.854} C_VEL
LIN {X 0,Y 136.527,Z 829.45,A -85,B 0,C 180,E1 -27882.668,E2 -27882.668} C_VEL
LIN {X 0,Y 126.746,Z 835.174,A -85,B 0,C 180,E1 -27885.55,E2 -27885.55} C_VEL
LIN {X 0,Y 115.987,Z 840.148,A -85,B 0,C 180,E1 -27889.526,E2 -27889.526} C_VEL
LIN {X 0,Y 105.923,Z 843.687,A -85,B 0,C 180,E1 -27894.39,E2 -27894.39} C_VEL
LIN {X 0,Y 97.251,Z 845.733,A -85,B 0,C 180,E1 -27899.999,E2 -27899.999} C_VEL
LIN {X 0,Y 92.986,Z 846.275,A -85,B 0,C 180,E1 -27903.543,E2 -27903.543} C_VEL
LIN {X 0,Y 89.259,Z 846.58,A -85,B 0,C 180,E1 -27906.414,E2 -27906.414} C_VEL
LIN {X 0,Y 82.137,Z 846.417,A -85,B 0,C 180,E1 -27911.021,E2 -27911.021} C_VEL
LIN {X 0,Y 76.773,Z 845.702,A -85,B 0,C 180,E1 -27915.222,E2 -27915.222} C_VEL
LIN {X 0,Y 73.739,Z 844.846,A -85,B 0,C 180,E1 -27919.036,E2 -27919.036} C_VEL
LIN {X 0,Y 73.046,Z 844.469,A -85,B 0,C 180,E1 -27920.453,E2 -27920.453} C_VEL
LIN {X 0,Y 70.171,Z 841.725,A -85,B 0,C 180,E1 -27930.05,E2 -27930.05} C_VEL
LIN {X 0,Y 69.145,Z 837.234,A -85,B 0,C 180,E1 -27941.122,E2 -27941.122} C_VEL
LIN {X 0,Y 70.038,Z 831.8,A -85,B 0,C 180,E1 -27951.047,E2 -27951.047} C_VEL
LIN {X 0,Y 71.873,Z 825.964,A -85,B 0,C 180,E1 -27959.119,E2 -27959.119} C_VEL
LIN {X 0,Y 74.584,Z 819.167,A -85,B 0,C 180,E1 -27966.396,E2 -27966.396} C_VEL
LIN {X 0,Y 78.107,Z 811.084,A -85,B 0,C 180,E1 -27972.999,E2 -27972.999} C_VEL
LIN {X 0,Y 82.497,Z 801.291,A -85,B 0,C 180,E1 -27978.952,E2 -27978.952} C_VEL
LIN {X 0,Y 86.947,Z 790.904,A -85,B 0,C 180,E1 -27983.621,E2 -27983.621} C_VEL
LIN {X 0,Y 89.429,Z 784.078,A -85,B 0,C 180,E1 -27986.059,E2 -27986.059} C_VEL
LIN {X 0,Y 90.39,Z 773.544,A -85,B 0,C 180,E1 -27990.002,E2 -27990.002} C_VEL
LIN {X 0,Y 90.977,Z 761.249,A -85,B 0,C 180,E1 -27993.849,E2 -27993.849} C_VEL
LIN {X 0,Y 90.816,Z 759.395,A -85,B 0,C 180,E1 -27994.441,E2 -27994.441} C_VEL
LIN {X 0,Y 85.012,Z 759.775,A -85,B 0,C 180,E1 -27997.235,E2 -27997.235} C_VEL
LIN {X 0,Y 80.567,Z 758.91,A -85,B 0,C 180,E1 -28000.05,E2 -28000.05} C_VEL
LIN {X 0,Y 80.061,Z 758.041,A -85,B 0,C 180,E1 -28000.649,E2 -28000.649} C_VEL
LIN {X 0,Y 76.566,Z 765.428,A -85,B 0,C 180,E1 -28008.631,E2 -28008.631} C_VEL
LIN {X 0,Y 74.743,Z 769.975,A -85,B 0,C 180,E1 -28015.035,E2 -28015.035} C_VEL
LIN {X 0,Y 73.584,Z 775.42,A -85,B 0,C 180,E1 -28024.967,E2 -28024.967} C_VEL
LIN {X 0,Y 74.537,Z 779.348,A -85,B 0,C 180,E1 -28035.008,E2 -28035.008} C_VEL
LIN {X 0,Y 77.538,Z 781.962,A -85,B 0,C 180,E1 -28044.666,E2 -28044.666} C_VEL
LIN {X 0,Y 80.584,Z 782.996,A -85,B 0,C 180,E1 -28050.712,E2 -28050.712} C_VEL
LIN {X 0,Y 84.435,Z 783.418,A -85,B 0,C 180,E1 -28056.295,E2 -28056.295} C_VEL
LIN {X 0,Y 89.19,Z 783.23,A -85,B 0,C 180,E1 -28061.628,E2 -28061.628} C_VEL
LIN {X 0,Y 95.613,Z 782.183,A -85,B 0,C 180,E1 -28067.261,E2 -28067.261} C_VEL
LIN {X 0,Y 102.724,Z 780.216,A -85,B 0,C 180,E1 -28072.136,E2 -28072.136} C_VEL
LIN {X 0,Y 112.569,Z 776.289,A -85,B 0,C 180,E1 -28077.379,E2 -28077.379} C_VEL
LIN {X 0,Y 118.076,Z 773.54,A -85,B 0,C 180,E1 -28080.001,E2 -28080.001} C_VEL
LIN {X 0,Y 120.243,Z 772.227,A -85,B 0,C 180,E1 -28083.351,E2 -28083.351} C_VEL
LIN {X 0,Y 121.977,Z 771.191,A -85,B 0,C 180,E1 -28086.618,E2 -28086.618} C_VEL
LIN {X 0,Y 122.619,Z 771.02,A -85,B 0,C 180,E1 -28089.902,E2 -28089.902} C_VEL
LIN {X 0,Y 122.118,Z 771.828,A -85,B 0,C 180,E1 -28093.31,E2 -28093.31} C_VEL
LIN {X 0,Y 121.526,Z 773.021,A -85,B 0,C 180,E1 -28096.808,E2 -28096.808} C_VEL
LIN {X 0,Y 120.724,Z 775.089,A -85,B 0,C 180,E1 -28101.335,E2 -28101.335} C_VEL
LIN {X 0,Y 119.743,Z 776.904,A -85,B 0,C 180,E1 -28104.259,E2 -28104.259} C_VEL
LIN {X 0,Y 119.219,Z 777.624,A -85,B 0,C 180,E1 -28105.161,E2 -28105.161} C_VEL
LIN {X 0,Y 114.986,Z 781.016,A -85,B 0,C 180,E1 -28107.592,E2 -28107.592} C_VEL
LIN {X 0,Y 107.405,Z 786.29,A -85,B 0,C 180,E1 -28111.715,E2 -28111.715} C_VEL
LIN {X 0,Y 99.986,Z 790.703,A -85,B 0,C 180,E1 -28116.064,E2 -28116.064} C_VEL
LIN {X 0,Y 93.087,Z 794.219,A -85,B 0,C 180,E1 -28120.972,E2 -28120.972} C_VEL
LIN {X 0,Y 85.405,Z 797.718,A -85,B 0,C 180,E1 -28128.256,E2 -28128.256} C_VEL
LIN {X 0,Y 81.418,Z 807.182,A -85,B 0,C 180,E1 -28132.823,E2 -28132.823} C_VEL
LIN {X 0,Y 77.432,Z 816.11,A -85,B 0,C 180,E1 -28138.538,E2 -28138.538} C_VEL
LIN {X 0,Y 73.741,Z 824.802,A -85,B 0,C 180,E1 -28146.103,E2 -28146.103} C_VEL
LIN {X 0,Y 71.371,Z 831.829,A -85,B 0,C 180,E1 -28154.285,E2 -28154.285} C_VEL
LIN {X 0,Y 70.416,Z 836.573,A -85,B 0,C 180,E1 -28161.387,E2 -28161.387} C_VEL
LIN {X 0,Y 70.281,Z 841.115,A -85,B 0,C 180,E1 -28169.997,E2 -28169.997} C_VEL
LIN {X 0,Y 70.209,Z 843.446,A -85,B 0,C 180,E1 -28175.742,E2 -28175.742} C_VEL
LIN {X 0,Y 70.589,Z 845.319,A -85,B 0,C 180,E1 -28181.482,E2 -28181.482} C_VEL
LIN {X 0,Y 73.187,Z 847.9,A -85,B 0,C 180,E1 -28192.585,E2 -28192.585} C_VEL
LIN {X 0,Y 78.344,Z 849.124,A -85,B 0,C 180,E1 -28202.561,E2 -28202.561} C_VEL
LIN {X 0,Y 85.777,Z 849.017,A -85,B 0,C 180,E1 -28210.952,E2 -28210.952} C_VEL
LIN {X 0,Y 94.854,Z 847.517,A -85,B 0,C 180,E1 -28217.807,E2 -28217.807} C_VEL
LIN {X 0,Y 105.125,Z 844.682,A -85,B 0,C 180,E1 -28223.341,E2 -28223.341} C_VEL
LIN {X 0,Y 116.244,Z 840.416,A -85,B 0,C 180,E1 -28227.821,E2 -28227.821} C_VEL
LIN {X 0,Y 128.277,Z 834.439,A -85,B 0,C 180,E1 -28231.231,E2 -28231.231} C_VEL
LIN {X 0,Y 139.123,Z 827.76,A -85,B 0,C 180,E1 -28233.719,E2 -28233.719} C_VEL
LIN {X 0,Y 146.826,Z 822.068,A -85,B 0,C 180,E1 -28235.426,E2 -28235.426} C_VEL
LIN {X 0,Y 147.505,Z 821.491,A -85,B 0,C 180,E1 -28236.108,E2 -28236.108} C_VEL
LIN {X 0,Y 145.517,Z 822.969,A -85,B 0,C 180,E1 -28237.27,E2 -28237.27} C_VEL
LIN {X 0,Y 136.336,Z 829.245,A -85,B 0,C 180,E1 -28239.358,E2 -28239.358} C_VEL
LIN {X 0,Y 125.525,Z 835.339,A -85,B 0,C 180,E1 -28242.133,E2 -28242.133} C_VEL
LIN {X 0,Y 114.283,Z 840.305,A -85,B 0,C 180,E1 -28245.759,E2 -28245.759} C_VEL
LIN {X 0,Y 107.113,Z 842.826,A -85,B 0,C 180,E1 -28248.647,E2 -28248.647} C_VEL
LIN {X 0,Y 99.215,Z 844.932,A -85,B 0,C 180,E1 -28252.593,E2 -28252.593} C_VEL
LIN {X 0,Y 91.444,Z 846.305,A -85,B 0,C 180,E1 -28257.541,E2 -28257.541} C_VEL
LIN {X 0,Y 83.12,Z 846.793,A -85,B 0,C 180,E1 -28264.85,E2 -28264.85} C_VEL
LIN {X 0,Y 78.587,Z 846.357,A -85,B 0,C 180,E1 -28270.368,E2 -28270.368} C_VEL
LIN {X 0,Y 74.006,Z 845.009,A -85,B 0,C 180,E1 -28278.269,E2 -28278.269} C_VEL
LIN {X 0,Y 73.046,Z 844.469,A -85,B 0,C 180,E1 -28280.453,E2 -28280.453} C_VEL
LIN {X 0,Y 70.834,Z 843.33,A -85,B 0,C 180,E1 -28284.705,E2 -28284.705} C_VEL
LIN {X 0,Y 66.304,Z 840.687,A -85,B 0,C 180,E1 -28291.745,E2 -28291.745} C_VEL
LIN {X 0,Y 63.263,Z 838.019,A -85,B 0,C 180,E1 -28297.859,E2 -28297.859} C_VEL
LIN {X 0,Y 62.208,Z 835.721,A -85,B 0,C 180,E1 -28302.8,E2 -28302.8} C_VEL
LIN {X 0,Y 62.21,Z 834.906,A -85,B 0,C 180,E1 -28304.479,E2 -28304.479} C_VEL
LIN {X 0,Y 63.464,Z 829.605,A -85,B 0,C 180,E1 -28314.039,E2 -28314.039} C_VEL
LIN {X 0,Y 66.132,Z 822.443,A -85,B 0,C 180,E1 -28323.822,E2 -28323.822} C_VEL
LIN {X 0,Y 70.082,Z 813.643,A -85,B 0,C 180,E1 -28332.495,E2 -28332.495} C_VEL
LIN {X 0,Y 74.459,Z 804.408,A -85,B 0,C 180,E1 -28339.122,E2 -28339.122} C_VEL
LIN {X 0,Y 79.23,Z 794.055,A -85,B 0,C 180,E1 -28344.493,E2 -28344.493} C_VEL
LIN {X 0,Y 83.102,Z 784.563,A -85,B 0,C 180,E1 -28348.185,E2 -28348.185} C_VEL
LIN {X 0,Y 84.461,Z 772.122,A -85,B 0,C 180,E1 -28353.129,E2 -28353.129} C_VEL
LIN {X 0,Y 84.885,Z 767.307,A -85,B 0,C 180,E1 -28354.752,E2 -28354.752} C_VEL
LIN {X 0,Y 84.687,Z 766.3,A -85,B 0,C 180,E1 -28355.226,E2 -28355.226} C_VEL
LIN {X 0,Y 78.283,Z 765.494,A -85,B 0,C 180,E1 -28359.057,E2 -28359.057} C_VEL
LIN {X 0,Y 75.252,Z 766.012,A -85,B 0,C 180,E1 -28360.768,E2 -28360.768} C_VEL
LIN {X 0,Y 72.146,Z 765.767,A -85,B 0,C 180,E1 -28363.064,E2 -28363.064} C_VEL
LIN {X 0,Y 70.534,Z 764.219,A -85,B 0,C 180,E1 -28365.11,E2 -28365.11} C_VEL
LIN {X 0,Y 67.662,Z 770.674,A -85,B 0,C 180,E1 -28374.553,E2 -28374.553} C_VEL
LIN {X 0,Y 66.508,Z 776.231,A -85,B 0,C 180,E1 -28385.601,E2 -28385.601} C_VEL
LIN {X 0,Y 67.706,Z 780.246,A -85,B 0,C 180,E1 -28396.607,E2 -28396.607} C_VEL
LIN {X 0,Y 69.777,Z 782.19,A -85,B 0,C 180,E1 -28403.689,E2 -28403.689} C_VEL
LIN {X 0,Y 73.296,Z 783.712,A -85,B 0,C 180,E1 -28411.353,E2 -28411.353} C_VEL
LIN {X 0,Y 78.577,Z 784.497,A -85,B 0,C 180,E1 -28419.038,E2 -28419.038} C_VEL
LIN {X 0,Y 86.539,Z 784.163,A -85,B 0,C 180,E1 -28427.052,E2 -28427.052} C_VEL
LIN {X 0,Y 92.381,Z 783.145,A -85,B 0,C 180,E1 -28431.501,E2 -28431.501} C_VEL
LIN {X 0,Y 102.208,Z 780.394,A -85,B 0,C 180,E1 -28437.293,E2 -28437.293} C_VEL
LIN {X 0,Y 112.521,Z 776.19,A -85,B 0,C 180,E1 -28442.024,E2 -28442.024} C_VEL
LIN {X 0,Y 113.717,Z 775.634,A -85,B 0,C 180,E1 -28443.544,E2 -28443.544} C_VEL
LIN {X 0,Y 115.696,Z 774.747,A -85,B 0,C 180,E1 -28446.979,E2 -28446.979} C_VEL
LIN {X 0,Y 116.401,Z 774.742,A -85,B 0,C 180,E1 -28450.436,E2 -28450.436} C_VEL
LIN {X 0,Y 115.761,Z 775.732,A -85,B 0,C 180,E1 -28454.055,E2 -28454.055} C_VEL
LIN {X 0,Y 115.049,Z 777.076,A -85,B 0,C 180,E1 -28457.785,E2 -28457.785} C_VEL
LIN {X 0,Y 113.897,Z 779.18,A -85,B 0,C 180,E1 -28462.241,E2 -28462.241} C_VEL
LIN {X 0,Y 111.722,Z 781.044,A -85,B 0,C 180,E1 -28464.194,E2 -28464.194} C_VEL
LIN {X 0,Y 103.522,Z 786.205,A -85,B 0,C 180,E1 -28468.375,E2 -28468.375} C_VEL
LIN {X 0,Y 93.345,Z 791.484,A -85,B 0,C 180,E1 -28474.082,E2 -28474.082} C_VEL
LIN {X 0,Y 83.993,Z 795.427,A -85,B 0,C 180,E1 -28481.14,E2 -28481.14} C_VEL
LIN {X 0,Y 79.089,Z 797.194,A -85,B 0,C 180,E1 -28486.03,E2 -28486.03} C_VEL
LIN {X 0,Y 74.974,Z 806.485,A -85,B 0,C 180,E1 -28490.744,E2 -28490.744} C_VEL
LIN {X 0,Y 70.721,Z 815.503,A -85,B 0,C 180,E1 -28496.864,E2 -28496.864} C_VEL
LIN {X 0,Y 66.772,Z 824.266,A -85,B 0,C 180,E1 -28505.098,E2 -28505.098} C_VEL
LIN {X 0,Y 64.284,Z 831.345,A -85,B 0,C 180,E1 -28514.135,E2 -28514.135} C_VEL
LIN {X 0,Y 63.241,Z 836.964,A -85,B 0,C 180,E1 -28523.616,E2 -28523.616} C_VEL
LIN {X 0,Y 63.277,Z 840.653,A -85,B 0,C 180,E1 -28531.587,E2 -28531.587} C_VEL
LIN {X 0,Y 63.692,Z 844.429,A -85,B 0,C 180,E1 -28542.746,E2 -28542.746} C_VEL
LIN {X 0,Y 66.685,Z 847.306,A -85,B 0,C 180,E1 -28554.93,E2 -28554.93} C_VEL
LIN {X 0,Y 72.464,Z 848.75,A -85,B 0,C 180,E1 -28565.582,E2 -28565.582} C_VEL
LIN {X 0,Y 80.544,Z 848.883,A -85,B 0,C 180,E1 -28574.267,E2 -28574.267} C_VEL
LIN {X 0,Y 90.229,Z 847.706,A -85,B 0,C 180,E1 -28581.156,E2 -28581.156} C_VEL
LIN {X 0,Y 101.054,Z 845.161,A -85,B 0,C 180,E1 -28586.566,E2 -28586.566} C_VEL
LIN {X 0,Y 112.659,Z 841.207,A -85,B 0,C 180,E1 -28590.847,E2 -28590.847} C_VEL
LIN {X 0,Y 125.06,Z 835.676,A -85,B 0,C 180,E1 -28594.042,E2 -28594.042} C_VEL
LIN {X 0,Y 131.426,Z 832.197,A -85,B 0,C 180,E1 -28595.373,E2 -28595.373} C_VEL
LIN {X 0,Y 134.162,Z 830.562,A -85,B 0,C 180,E1 -28596.553,E2 -28596.553} C_VEL
LIN {X 0,Y 125.037,Z 835.448,A -85,B 0,C 180,E1 -28598.57,E2 -28598.57} C_VEL
LIN {X 0,Y 113.123,Z 840.483,A -85,B 0,C 180,E1 -28601.902,E2 -28601.902} C_VEL
LIN {X 0,Y 101.288,Z 844.164,A -85,B 0,C 180,E1 -28606.255,E2 -28606.255} C_VEL
LIN {X 0,Y 91.445,Z 846.167,A -85,B 0,C 180,E1 -28611.157,E2 -28611.157} C_VEL
LIN {X 0,Y 84.576,Z 846.889,A -85,B 0,C 180,E1 -28615.644,E2 -28615.644} C_VEL
LIN {X 0,Y 77.347,Z 846.931,A -85,B 0,C 180,E1 -28621.915,E2 -28621.915} C_VEL
LIN {X 0,Y 69.828,Z 845.706,A -85,B 0,C 180,E1 -28631.612,E2 -28631.612} C_VEL
LIN {X 0,Y 64.976,Z 843.227,A -85,B 0,C 180,E1 -28642.244,E2 -28642.244} C_VEL
LIN {X 0,Y 62.44,Z 839.303,A -85,B 0,C 180,E1 -28654.247,E2 -28654.247} C_VEL
LIN {X 0,Y 62.21,Z 834.906,A -85,B 0,C 180,E1 -28664.479,E2 -28664.479} C_VEL
LIN {X 0,Y 62.173,Z 833.232,A -85,B 0,C 180,E1 -28667.759,E2 -28667.759} C_VEL
LIN {X 0,Y 61.485,Z 830.453,A -85,B 0,C 180,E1 -28672.573,E2 -28672.573} C_VEL
LIN {X 0,Y 59.833,Z 823.001,A -85,B 0,C 180,E1 -28683.683,E2 -28683.683} C_VEL
LIN {X 0,Y 60.419,Z 819.42,A -85,B 0,C 180,E1 -28688.209,E2 -28688.209} C_VEL
LIN {X 0,Y 60.928,Z 818.162,A -85,B 0,C 180,E1 -28689.601,E2 -28689.601} C_VEL
LIN {X 0,Y 65.195,Z 809.602,A -85,B 0,C 180,E1 -28697.553,E2 -28697.553} C_VEL
LIN {X 0,Y 70.31,Z 799.488,A -85,B 0,C 180,E1 -28704.266,E2 -28704.266} C_VEL
LIN {X 0,Y 75.41,Z 788.58,A -85,B 0,C 180,E1 -28709.335,E2 -28709.335} C_VEL
LIN {X 0,Y 76.842,Z 785.192,A -85,B 0,C 180,E1 -28710.611,E2 -28710.611} C_VEL
LIN {X 0,Y 78.344,Z 774.625,A -85,B 0,C 180,E1 -28715.149,E2 -28715.149} C_VEL
LIN {X 0,Y 78.465,Z 773.39,A -85,B 0,C 180,E1 -28715.642,E2 -28715.642} C_VEL
LIN {X 0,Y 77.815,Z 772.169,A -85,B 0,C 180,E1 -28716.552,E2 -28716.552} C_VEL
LIN {X 0,Y 69.882,Z 772.224,A -85,B 0,C 180,E1 -28721.607,E2 -28721.607} C_VEL
LIN {X 0,Y 65.6,Z 771.595,A -85,B 0,C 180,E1 -28725.38,E2 -28725.38} C_VEL
LIN {X 0,Y 61.615,Z 770.184,A -85,B 0,C 180,E1 -28730.014,E2 -28730.014} C_VEL
LIN {X 0,Y 61.253,Z 769.691,A -85,B 0,C 180,E1 -28730.981,E2 -28730.981} C_VEL
LIN {X 0,Y 59.59,Z 774.822,A -85,B 0,C 180,E1 -28741.054,E2 -28741.054} C_VEL
LIN {X 0,Y 60.159,Z 779.887,A -85,B 0,C 180,E1 -28754.507,E2 -28754.507} C_VEL
LIN {X 0,Y 63.34,Z 783.109,A -85,B 0,C 180,E1 -28766.305,E2 -28766.305} C_VEL
LIN {X 0,Y 68.814,Z 785.062,A -85,B 0,C 180,E1 -28776.813,E2 -28776.813} C_VEL
LIN {X 0,Y 74.048,Z 785.626,A -85,B 0,C 180,E1 -28783.458,E2 -28783.458} C_VEL
LIN {X 0,Y 81.07,Z 785.42,A -85,B 0,C 180,E1 -28790.016,E2 -28790.016} C_VEL
LIN {X 0,Y 91.488,Z 783.755,A -85,B 0,C 180,E1 -28797.055,E2 -28797.055} C_VEL
LIN {X 0,Y 101.985,Z 780.672,A -85,B 0,C 180,E1 -28802.209,E2 -28802.209} C_VEL
LIN {X 0,Y 105.86,Z 779.229,A -85,B 0,C 180,E1 -28803.807,E2 -28803.807} C_VEL
LIN {X 0,Y 109.239,Z 778.008,A -85,B 0,C 180,E1 -28807.393,E2 -28807.393} C_VEL
LIN {X 0,Y 109.874,Z 778.199,A -85,B 0,C 180,E1 -28811.064,E2 -28811.064} C_VEL
LIN {X 0,Y 109.128,Z 779.317,A -85,B 0,C 180,E1 -28814.972,E2 -28814.972} C_VEL
LIN {X 0,Y 108.207,Z 780.821,A -85,B 0,C 180,E1 -28818.951,E2 -28818.951} C_VEL
LIN {X 0,Y 106.055,Z 782.748,A -85,B 0,C 180,E1 -28821.909,E2 -28821.909} C_VEL
LIN {X 0,Y 97.173,Z 787.53,A -85,B 0,C 180,E1 -28826.201,E2 -28826.201} C_VEL
LIN {X 0,Y 86.855,Z 792.051,A -85,B 0,C 180,E1 -28831.826,E2 -28831.826} C_VEL
LIN {X 0,Y 75.773,Z 795.794,A -85,B 0,C 180,E1 -28840.487,E2 -28840.487} C_VEL
LIN {X 0,Y 72.911,Z 796.708,A -85,B 0,C 180,E1 -28843.448,E2 -28843.448} C_VEL
LIN {X 0,Y 68.634,Z 805.781,A -85,B 0,C 180,E1 -28848.269,E2 -28848.269} C_VEL
LIN {X 0,Y 64.069,Z 814.834,A -85,B 0,C 180,E1 -28854.834,E2 -28854.834} C_VEL
LIN {X 0,Y 60.451,Z 822.334,A -85,B 0,C 180,E1 -28862.284,E2 -28862.284} C_VEL
LIN {X 0,Y 57.511,Z 829.69,A -85,B 0,C 180,E1 -28872.208,E2 -28872.208} C_VEL
LIN {X 0,Y 56.254,Z 835.58,A -85,B 0,C 180,E1 -28882.819,E2 -28882.819} C_VEL
LIN {X 0,Y 56.264,Z 839.647,A -85,B 0,C 180,E1 -28892.138,E2 -28892.138} C_VEL
LIN {X 0,Y 56.836,Z 843.518,A -85,B 0,C 180,E1 -28904.314,E2 -28904.314} C_VEL
LIN {X 0,Y 60.34,Z 846.591,A -85,B 0,C 180,E1 -28917.764,E2 -28917.764} C_VEL
LIN {X 0,Y 66.824,Z 848.329,A -85,B 0,C 180,E1 -28929.122,E2 -28929.122} C_VEL
LIN {X 0,Y 75.619,Z 848.743,A -85,B 0,C 180,E1 -28938.027,E2 -28938.027} C_VEL
LIN {X 0,Y 85.947,Z 847.813,A -85,B 0,C 180,E1 -28944.851,E2 -28944.851} C_VEL
